Yaskawa INFORM job: A_ROOF_SIDE_0617_2_PAINT_42.JBI

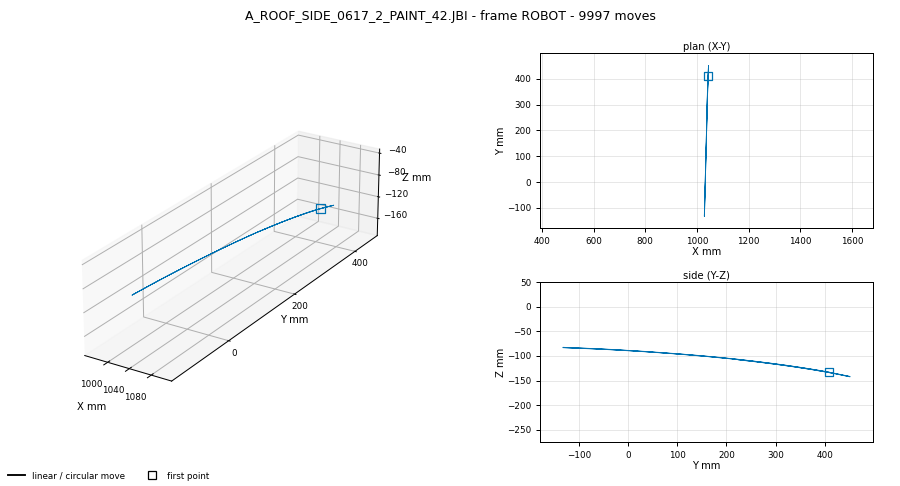
[picture p0: tool path of A_ROOF_SIDE_0617_2_PAINT_42.JBI in frame ROBOT, 9997 of 9997 moves have a stored position in this frame; points joined in program order, loops and branches not executed]
/JOB
//NAME A_ROOF_SIDE_0617_2_PAINT42
//POS
///NPOS 9997,0,0,0,0,0
///TOOL 1
///USER 0
///POSTYPE ROBOT
///RECTAN
///RCONF 1,0,0,0,0,0,0,0,0,0,0,0,0,0,0,0,0,0,0,0,0,0,0,0
C00000=1043.700,409.067,-132.998,174.418,43.875,158.706
C00001=1043.690,408.820,-132.952,174.408,43.868,158.704
C00002=1043.680,408.575,-132.906,174.398,43.862,158.701
C00003=1043.671,408.330,-132.861,174.389,43.855,158.699
C00004=1043.661,408.085,-132.816,174.379,43.848,158.696
C00005=1043.651,407.839,-132.770,174.370,43.842,158.694
C00006=1043.642,407.593,-132.725,174.361,43.835,158.691
C00007=1043.632,407.347,-132.680,174.352,43.829,158.689
C00008=1043.623,407.101,-132.635,174.342,43.822,158.686
C00009=1043.613,406.855,-132.589,174.333,43.816,158.684
C00010=1043.603,406.610,-132.544,174.325,43.809,158.681
C00011=1043.594,406.364,-132.499,174.315,43.802,158.679
C00012=1043.586,406.155,-132.460,174.308,43.797,158.677
C00013=1043.578,405.946,-132.422,174.300,43.791,158.674
C00014=1043.570,405.736,-132.384,174.292,43.786,158.672
C00015=1043.561,405.527,-132.345,174.284,43.780,158.670
C00016=1043.554,405.317,-132.307,174.277,43.775,158.668
C00017=1043.545,405.108,-132.268,174.269,43.770,158.666
C00018=1043.537,404.898,-132.230,174.261,43.764,158.664
C00019=1043.530,404.689,-132.192,174.254,43.759,158.662
C00020=1043.520,404.444,-132.147,174.244,43.753,158.660
C00021=1043.511,404.197,-132.102,174.235,43.746,158.657
C00022=1043.502,403.952,-132.058,174.226,43.740,158.655
C00023=1043.492,403.706,-132.013,174.218,43.733,158.652
C00024=1043.483,403.460,-131.968,174.209,43.727,158.650
C00025=1043.474,403.214,-131.923,174.200,43.721,158.648
C00026=1043.464,402.968,-131.879,174.191,43.715,158.645
C00027=1043.454,402.723,-131.834,174.183,43.708,158.643
C00028=1043.445,402.477,-131.790,174.174,43.702,158.640
C00029=1043.436,402.231,-131.745,174.164,43.696,158.638
C00030=1043.427,401.985,-131.701,174.156,43.690,158.636
C00031=1043.417,401.740,-131.656,174.147,43.684,158.634
C00032=1043.408,401.494,-131.612,174.138,43.678,158.631
C00033=1043.399,401.248,-131.568,174.130,43.671,158.629
C00034=1043.390,401.002,-131.524,174.121,43.666,158.627
C00035=1043.380,400.757,-131.479,174.112,43.660,158.624
C00036=1043.371,400.511,-131.435,174.104,43.653,158.622
C00037=1043.362,400.264,-131.391,174.096,43.648,158.620
C00038=1043.353,400.019,-131.347,174.086,43.641,158.617
C00039=1043.344,399.773,-131.303,174.079,43.635,158.615
C00040=1043.334,399.527,-131.259,174.070,43.630,158.613
C00041=1043.325,399.281,-131.215,174.062,43.623,158.611
C00042=1043.315,399.035,-131.171,174.053,43.618,158.609
C00043=1043.306,398.789,-131.127,174.045,43.612,158.606
C00044=1043.297,398.544,-131.083,174.036,43.606,158.604
C00045=1043.288,398.297,-131.040,174.028,43.600,158.602
C00046=1043.279,398.051,-130.996,174.019,43.594,158.600
C00047=1043.270,397.805,-130.952,174.012,43.588,158.598
C00048=1043.261,397.560,-130.908,174.003,43.583,158.595
C00049=1043.252,397.313,-130.865,173.995,43.577,158.593
C00050=1043.243,397.068,-130.821,173.986,43.571,158.591
C00051=1043.234,396.822,-130.777,173.978,43.565,158.589
C00052=1043.225,396.575,-130.734,173.970,43.559,158.587
C00053=1043.216,396.329,-130.690,173.962,43.554,158.584
C00054=1043.206,396.084,-130.647,173.953,43.548,158.582
C00055=1043.198,395.838,-130.604,173.945,43.542,158.580
C00056=1043.188,395.592,-130.560,173.937,43.536,158.578
C00057=1043.180,395.346,-130.517,173.929,43.531,158.576
C00058=1043.171,395.100,-130.474,173.921,43.525,158.574
C00059=1043.162,394.854,-130.430,173.913,43.519,158.572
C00060=1043.153,394.608,-130.387,173.905,43.514,158.570
C00061=1043.144,394.362,-130.344,173.897,43.508,158.568
C00062=1043.135,394.116,-130.300,173.889,43.502,158.565
C00063=1043.126,393.870,-130.258,173.880,43.497,158.563
C00064=1043.117,393.624,-130.215,173.873,43.491,158.561
C00065=1043.109,393.378,-130.172,173.865,43.486,158.559
C00066=1043.100,393.131,-130.128,173.856,43.480,158.557
C00067=1043.090,392.886,-130.086,173.849,43.475,158.555
C00068=1043.082,392.639,-130.043,173.841,43.469,158.553
C00069=1043.073,392.393,-130.000,173.833,43.464,158.551
C00070=1043.064,392.148,-129.957,173.825,43.458,158.549
C00071=1043.056,391.902,-129.914,173.817,43.453,158.547
C00072=1043.041,391.502,-129.844,173.805,43.444,158.544
C00073=1043.027,391.102,-129.775,173.792,43.435,158.540
C00074=1043.012,390.702,-129.706,173.780,43.426,158.537
C00075=1042.998,390.303,-129.637,173.767,43.418,158.534
C00076=1042.989,390.057,-129.594,173.759,43.413,158.532
C00077=1042.981,389.811,-129.551,173.752,43.407,158.530
C00078=1042.972,389.565,-129.509,173.744,43.402,158.528
C00079=1042.963,389.319,-129.466,173.737,43.397,158.526
C00080=1042.954,389.073,-129.424,173.729,43.391,158.524
C00081=1042.946,388.826,-129.381,173.722,43.386,158.522
C00082=1042.937,388.580,-129.339,173.713,43.381,158.520
C00083=1042.929,388.334,-129.297,173.706,43.376,158.519
C00084=1042.919,388.088,-129.254,173.698,43.371,158.517
C00085=1042.910,387.842,-129.213,173.691,43.365,158.515
C00086=1042.902,387.595,-129.170,173.683,43.360,158.513
C00087=1042.893,387.349,-129.128,173.676,43.355,158.511
C00088=1042.884,387.103,-129.086,173.669,43.350,158.509
C00089=1042.876,386.856,-129.044,173.661,43.345,158.507
C00090=1042.867,386.610,-129.002,173.654,43.340,158.505
C00091=1042.859,386.364,-128.961,173.646,43.334,158.503
C00092=1042.849,386.118,-128.918,173.639,43.330,158.502
C00093=1042.841,385.872,-128.876,173.632,43.324,158.500
C00094=1042.832,385.625,-128.834,173.624,43.319,158.498
C00095=1042.823,385.379,-128.793,173.617,43.315,158.496
C00096=1042.815,385.133,-128.751,173.609,43.309,158.494
C00097=1042.807,384.887,-128.709,173.602,43.304,158.492
C00098=1042.798,384.640,-128.667,173.595,43.300,158.490
C00099=1042.789,384.394,-128.625,173.588,43.295,158.489
C00100=1042.781,384.148,-128.584,173.580,43.289,158.487
C00101=1042.772,383.902,-128.542,173.573,43.284,158.485
C00102=1042.763,383.655,-128.500,173.566,43.280,158.483
C00103=1042.755,383.409,-128.459,173.558,43.275,158.481
C00104=1042.746,383.163,-128.418,173.551,43.270,158.480
C00105=1042.738,382.916,-128.375,173.545,43.265,158.478
C00106=1042.730,382.670,-128.334,173.538,43.260,158.476
C00107=1042.721,382.423,-128.293,173.530,43.255,158.474
C00108=1042.712,382.177,-128.251,173.523,43.250,158.472
C00109=1042.705,381.931,-128.209,173.516,43.245,158.471
C00110=1042.696,381.684,-128.168,173.508,43.241,158.469
C00111=1042.688,381.438,-128.127,173.501,43.236,158.467
C00112=1042.679,381.192,-128.085,173.495,43.231,158.465
C00113=1042.672,380.945,-128.044,173.488,43.226,158.464
C00114=1042.663,380.699,-128.002,173.480,43.221,158.462
C00115=1042.655,380.453,-127.962,173.473,43.217,158.460
C00116=1042.646,380.206,-127.920,173.466,43.212,158.458
C00117=1042.638,379.960,-127.879,173.460,43.207,158.457
C00118=1042.629,379.713,-127.837,173.453,43.202,158.455
C00119=1042.621,379.467,-127.797,173.446,43.198,158.453
C00120=1042.613,379.221,-127.756,173.438,43.193,158.451
C00121=1042.604,378.974,-127.714,173.432,43.188,158.450
C00122=1042.596,378.728,-127.674,173.425,43.183,158.448
C00123=1042.588,378.481,-127.633,173.418,43.178,158.446
C00124=1042.580,378.235,-127.592,173.411,43.174,158.445
C00125=1042.571,377.988,-127.551,173.405,43.170,158.443
C00126=1042.563,377.742,-127.510,173.398,43.165,158.441
C00127=1042.555,377.495,-127.470,173.391,43.160,158.440
C00128=1042.542,377.130,-127.409,173.380,43.154,158.437
C00129=1042.530,376.764,-127.349,173.370,43.147,158.435
C00130=1042.518,376.398,-127.288,173.360,43.140,158.432
C00131=1042.505,376.032,-127.228,173.351,43.133,158.430
C00132=1042.497,375.786,-127.187,173.344,43.128,158.428
C00133=1042.489,375.539,-127.146,173.337,43.124,158.427
C00134=1042.481,375.292,-127.106,173.331,43.120,158.425
C00135=1042.472,375.046,-127.066,173.324,43.115,158.423
C00136=1042.464,374.799,-127.026,173.317,43.111,158.422
C00137=1042.456,374.552,-126.985,173.311,43.106,158.420
C00138=1042.448,374.306,-126.944,173.304,43.102,158.419
C00139=1042.440,374.059,-126.904,173.298,43.098,158.417
C00140=1042.432,373.813,-126.863,173.291,43.093,158.416
C00141=1042.424,373.567,-126.823,173.284,43.089,158.414
C00142=1042.415,373.319,-126.783,173.278,43.084,158.412
C00143=1042.407,373.073,-126.743,173.271,43.080,158.411
C00144=1042.399,372.827,-126.702,173.265,43.076,158.409
C00145=1042.391,372.580,-126.662,173.258,43.071,158.408
C00146=1042.383,372.334,-126.621,173.252,43.067,158.406
C00147=1042.375,372.087,-126.581,173.245,43.062,158.404
C00148=1042.367,371.840,-126.541,173.239,43.058,158.403
C00149=1042.359,371.594,-126.501,173.232,43.054,158.401
C00150=1042.351,371.348,-126.461,173.226,43.050,158.400
C00151=1042.343,371.101,-126.421,173.219,43.045,158.398
C00152=1042.335,370.854,-126.381,173.213,43.041,158.397
C00153=1042.327,370.608,-126.340,173.206,43.037,158.395
C00154=1042.319,370.361,-126.301,173.200,43.032,158.394
C00155=1042.311,370.114,-126.261,173.193,43.028,158.392
C00156=1042.303,369.867,-126.222,173.188,43.024,158.391
C00157=1042.295,369.621,-126.182,173.181,43.020,158.389
C00158=1042.286,369.375,-126.142,173.175,43.016,158.388
C00159=1042.278,369.128,-126.102,173.169,43.011,158.386
C00160=1042.270,368.881,-126.063,173.162,43.007,158.385
C00161=1042.262,368.634,-126.023,173.156,43.003,158.383
C00162=1042.254,368.388,-125.983,173.149,42.999,158.382
C00163=1042.246,368.141,-125.943,173.144,42.995,158.380
C00164=1042.238,367.894,-125.904,173.137,42.991,158.379
C00165=1042.230,367.647,-125.864,173.131,42.987,158.377
C00166=1042.221,367.401,-125.825,173.125,42.983,158.376
C00167=1042.214,367.154,-125.785,173.118,42.978,158.374
C00168=1042.206,366.907,-125.747,173.112,42.974,158.373
C00169=1042.198,366.660,-125.707,173.107,42.970,158.371
C00170=1042.190,366.414,-125.667,173.100,42.966,158.370
C00171=1042.182,366.167,-125.628,173.094,42.962,158.368
C00172=1042.174,365.920,-125.588,173.088,42.958,158.367
C00173=1042.166,365.673,-125.548,173.081,42.954,158.366
C00174=1042.158,365.427,-125.510,173.076,42.950,158.364
C00175=1042.151,365.180,-125.470,173.070,42.946,158.363
C00176=1042.142,364.933,-125.431,173.063,42.942,158.361
C00177=1042.135,364.686,-125.392,173.057,42.938,158.360
C00178=1042.127,364.440,-125.353,173.051,42.934,158.358
C00179=1042.119,364.193,-125.313,173.045,42.930,158.357
C00180=1042.111,363.946,-125.274,173.039,42.926,158.356
C00181=1042.104,363.699,-125.235,173.033,42.922,158.354
C00182=1042.096,363.452,-125.196,173.027,42.918,158.353
C00183=1042.088,363.205,-125.156,173.021,42.914,158.351
C00184=1042.077,362.859,-125.102,173.012,42.909,158.349
C00185=1042.066,362.513,-125.047,173.004,42.904,158.348
C00186=1042.056,362.168,-124.992,172.997,42.898,158.346
C00187=1042.045,361.821,-124.938,172.988,42.893,158.344
C00188=1042.037,361.574,-124.899,172.981,42.889,158.342
C00189=1042.028,361.327,-124.860,172.976,42.885,158.341
C00190=1042.021,361.081,-124.822,172.970,42.881,158.340
C00191=1042.013,360.833,-124.782,172.964,42.877,158.338
C00192=1042.006,360.587,-124.744,172.959,42.873,158.337
C00193=1041.997,360.340,-124.705,172.952,42.870,158.335
C00194=1041.989,360.093,-124.666,172.946,42.866,158.334
C00195=1041.982,359.847,-124.628,172.941,42.862,158.333
C00196=1041.974,359.599,-124.589,172.935,42.859,158.332
C00197=1041.967,359.353,-124.550,172.929,42.855,158.330
C00198=1041.959,359.105,-124.512,172.923,42.851,158.329
C00199=1041.951,358.859,-124.474,172.917,42.847,158.328
C00200=1041.943,358.612,-124.435,172.911,42.843,158.326
C00201=1041.935,358.365,-124.397,172.906,42.840,158.325
C00202=1041.927,358.118,-124.358,172.900,42.836,158.324
C00203=1041.920,357.871,-124.320,172.895,42.833,158.322
C00204=1041.912,357.624,-124.281,172.889,42.829,158.321
C00205=1041.905,357.377,-124.242,172.883,42.825,158.320
C00206=1041.897,357.131,-124.204,172.877,42.822,158.318
C00207=1041.889,356.884,-124.166,172.871,42.818,158.317
C00208=1041.882,356.636,-124.128,172.866,42.814,158.316
C00209=1041.874,356.389,-124.089,172.860,42.810,158.314
C00210=1041.866,356.143,-124.051,172.854,42.807,158.313
C00211=1041.859,355.896,-124.013,172.849,42.803,158.312
C00212=1041.851,355.648,-123.975,172.843,42.800,158.311
C00213=1041.843,355.402,-123.937,172.838,42.796,158.309
C00214=1041.835,355.155,-123.898,172.832,42.793,158.308
C00215=1041.828,354.908,-123.861,172.827,42.789,158.307
C00216=1041.820,354.661,-123.822,172.821,42.786,158.306
C00217=1041.812,354.413,-123.785,172.816,42.782,158.305
C00218=1041.804,354.167,-123.747,172.810,42.779,158.303
C00219=1041.797,353.920,-123.709,172.804,42.775,158.302
C00220=1041.789,353.673,-123.671,172.799,42.771,158.301
C00221=1041.781,353.425,-123.633,172.792,42.768,158.299
C00222=1041.774,353.179,-123.595,172.787,42.765,158.298
C00223=1041.767,352.932,-123.557,172.781,42.761,158.297
C00224=1041.759,352.685,-123.519,172.776,42.758,158.296
C00225=1041.751,352.437,-123.481,172.771,42.754,158.295
C00226=1041.744,352.191,-123.443,172.766,42.751,158.293
C00227=1041.736,351.944,-123.406,172.760,42.747,158.292
C00228=1041.729,351.697,-123.368,172.755,42.744,158.291
C00229=1041.722,351.450,-123.330,172.749,42.740,158.290
C00230=1041.713,351.203,-123.293,172.744,42.737,158.288
C00231=1041.706,350.955,-123.255,172.738,42.733,158.287
C00232=1041.699,350.708,-123.217,172.733,42.730,158.286
C00233=1041.691,350.462,-123.179,172.727,42.726,158.285
C00234=1041.684,350.215,-123.142,172.722,42.723,158.284
C00235=1041.677,349.968,-123.104,172.717,42.720,158.283
C00236=1041.669,349.720,-123.067,172.711,42.717,158.281
C00237=1041.661,349.473,-123.029,172.706,42.713,158.280
C00238=1041.653,349.226,-122.992,172.700,42.710,158.279
C00239=1041.646,348.979,-122.954,172.695,42.706,158.278
C00240=1041.636,348.639,-122.903,172.688,42.702,158.276
C00241=1041.625,348.299,-122.852,172.681,42.697,158.275
C00242=1041.615,347.958,-122.800,172.673,42.693,158.273
C00243=1041.604,347.618,-122.749,172.666,42.688,158.271
C00244=1041.596,347.371,-122.712,172.660,42.685,158.270
C00245=1041.589,347.124,-122.674,172.655,42.682,158.269
C00246=1041.582,346.877,-122.637,172.650,42.679,158.268
C00247=1041.574,346.630,-122.600,172.644,42.675,158.267
C00248=1041.567,346.383,-122.562,172.640,42.672,158.266
C00249=1041.560,346.135,-122.526,172.634,42.669,158.264
C00250=1041.552,345.888,-122.489,172.629,42.666,158.263
C00251=1041.545,345.641,-122.451,172.624,42.662,158.262
C00252=1041.537,345.394,-122.414,172.618,42.659,158.261
C00253=1041.530,345.146,-122.377,172.613,42.656,158.260
C00254=1041.522,344.899,-122.340,172.609,42.653,158.259
C00255=1041.515,344.653,-122.303,172.603,42.649,158.258
C00256=1041.508,344.405,-122.266,172.598,42.646,158.257
C00257=1041.500,344.159,-122.229,172.592,42.643,158.255
C00258=1041.493,343.911,-122.192,172.587,42.640,158.254
C00259=1041.485,343.664,-122.156,172.583,42.637,158.253
C00260=1041.478,343.417,-122.118,172.577,42.634,158.252
C00261=1041.471,343.169,-122.081,172.572,42.631,158.251
C00262=1041.463,342.922,-122.044,172.567,42.628,158.250
C00263=1041.457,342.675,-122.008,172.562,42.624,158.249
C00264=1041.449,342.428,-121.971,172.557,42.621,158.248
C00265=1041.442,342.181,-121.934,172.552,42.618,158.247
C00266=1041.434,341.934,-121.897,172.546,42.615,158.245
C00267=1041.427,341.686,-121.861,172.542,42.612,158.244
C00268=1041.419,341.439,-121.824,172.537,42.609,158.243
C00269=1041.412,341.193,-121.788,172.532,42.606,158.242
C00270=1041.404,340.945,-121.752,172.526,42.603,158.241
C00271=1041.397,340.697,-121.715,172.522,42.599,158.240
C00272=1041.389,340.450,-121.678,172.517,42.596,158.239
C00273=1041.381,340.203,-121.642,172.511,42.594,158.238
C00274=1041.375,339.956,-121.605,172.506,42.591,158.237
C00275=1041.367,339.709,-121.569,172.502,42.588,158.236
C00276=1041.360,339.461,-121.533,172.496,42.585,158.235
C00277=1041.352,339.214,-121.496,172.491,42.582,158.234
C00278=1041.345,338.967,-121.459,172.487,42.579,158.233
C00279=1041.338,338.720,-121.423,172.482,42.576,158.232
C00280=1041.330,338.472,-121.387,172.476,42.573,158.231
C00281=1041.324,338.225,-121.350,172.472,42.570,158.230
C00282=1041.316,337.978,-121.314,172.467,42.567,158.229
C00283=1041.308,337.730,-121.278,172.462,42.564,158.228
C00284=1041.301,337.484,-121.242,172.457,42.561,158.227
C00285=1041.294,337.236,-121.205,172.452,42.558,158.225
C00286=1041.287,336.988,-121.169,172.447,42.555,158.224
C00287=1041.280,336.742,-121.133,172.443,42.552,158.223
C00288=1041.272,336.494,-121.097,172.437,42.549,158.222
C00289=1041.266,336.247,-121.061,172.432,42.546,158.221
C00290=1041.258,336.000,-121.024,172.428,42.543,158.220
C00291=1041.250,335.752,-120.988,172.423,42.540,158.219
C00292=1041.243,335.506,-120.952,172.419,42.538,158.218
C00293=1041.237,335.257,-120.916,172.413,42.535,158.217
C00294=1041.230,335.010,-120.880,172.408,42.532,158.216
C00295=1041.222,334.763,-120.844,172.404,42.529,158.215
C00296=1041.211,334.419,-120.795,172.397,42.525,158.214
C00297=1041.201,334.076,-120.745,172.390,42.521,158.212
C00298=1041.191,333.732,-120.695,172.384,42.517,158.211
C00299=1041.182,333.388,-120.645,172.377,42.514,158.210
C00300=1041.174,333.140,-120.609,172.372,42.511,158.209
C00301=1041.167,332.893,-120.574,172.368,42.507,158.208
C00302=1041.159,332.646,-120.537,172.363,42.505,158.207
C00303=1041.153,332.398,-120.502,172.357,42.502,158.206
C00304=1041.145,332.151,-120.466,172.353,42.499,158.205
C00305=1041.138,331.903,-120.431,172.348,42.497,158.204
C00306=1041.131,331.656,-120.395,172.344,42.494,158.203
C00307=1041.124,331.409,-120.359,172.339,42.491,158.202
C00308=1041.116,331.161,-120.323,172.335,42.488,158.201
C00309=1041.109,330.914,-120.288,172.329,42.485,158.200
C00310=1041.102,330.667,-120.252,172.325,42.483,158.199
C00311=1041.095,330.419,-120.217,172.320,42.480,158.198
C00312=1041.088,330.172,-120.181,172.316,42.477,158.197
C00313=1041.080,329.924,-120.145,172.311,42.474,158.196
C00314=1041.073,329.677,-120.110,172.307,42.472,158.195
C00315=1041.067,329.430,-120.074,172.302,42.469,158.194
C00316=1041.059,329.182,-120.040,172.297,42.467,158.193
C00317=1041.051,328.936,-120.004,172.292,42.464,158.192
C00318=1041.045,328.688,-119.969,172.288,42.461,158.192
C00319=1041.037,328.440,-119.933,172.283,42.459,158.191
C00320=1041.030,328.193,-119.899,172.279,42.456,158.190
C00321=1041.022,327.945,-119.863,172.274,42.453,158.189
C00322=1041.015,327.698,-119.828,172.270,42.451,158.188
C00323=1041.008,327.451,-119.793,172.265,42.448,158.187
C00324=1041.000,327.203,-119.757,172.261,42.445,158.186
C00325=1040.993,326.956,-119.723,172.256,42.443,158.185
C00326=1040.986,326.709,-119.687,172.251,42.440,158.184
C00327=1040.978,326.461,-119.653,172.246,42.438,158.183
C00328=1040.971,326.214,-119.617,172.242,42.435,158.182
C00329=1040.964,325.967,-119.583,172.237,42.433,158.181
C00330=1040.956,325.718,-119.547,172.233,42.430,158.181
C00331=1040.950,325.471,-119.512,172.228,42.428,158.180
C00332=1040.942,325.224,-119.478,172.224,42.425,158.179
C00333=1040.935,324.977,-119.443,172.219,42.423,158.178
C00334=1040.928,324.728,-119.408,172.215,42.420,158.177
C00335=1040.921,324.481,-119.373,172.211,42.417,158.176
C00336=1040.913,324.234,-119.339,172.206,42.415,158.175
C00337=1040.907,323.987,-119.304,172.202,42.412,158.174
C00338=1040.898,323.739,-119.269,172.197,42.410,158.173
C00339=1040.892,323.491,-119.234,172.193,42.408,158.173
C00340=1040.885,323.244,-119.198,172.188,42.405,158.172
C00341=1040.878,322.996,-119.165,172.184,42.403,158.171
C00342=1040.871,322.749,-119.129,172.180,42.400,158.170
C00343=1040.863,322.502,-119.095,172.174,42.398,158.169
C00344=1040.856,322.254,-119.059,172.170,42.395,158.168
C00345=1040.849,322.006,-119.026,172.166,42.392,158.167
C00346=1040.842,321.759,-118.990,172.161,42.390,158.166
C00347=1040.835,321.512,-118.956,172.157,42.387,158.166
C00348=1040.828,321.264,-118.921,172.152,42.385,158.165
C00349=1040.821,321.017,-118.887,172.148,42.382,158.164
C00350=1040.814,320.769,-118.852,172.144,42.380,158.163
C00351=1040.807,320.522,-118.818,172.139,42.377,158.162
C00352=1040.797,320.173,-118.768,172.134,42.374,158.161
C00353=1040.787,319.825,-118.720,172.127,42.370,158.160
C00354=1040.777,319.476,-118.671,172.121,42.367,158.158
C00355=1040.767,319.127,-118.623,172.115,42.363,158.157
C00356=1040.760,318.879,-118.588,172.110,42.362,158.156
C00357=1040.753,318.632,-118.554,172.106,42.359,158.156
C00358=1040.746,318.384,-118.519,172.102,42.357,158.155
C00359=1040.739,318.137,-118.485,172.097,42.354,158.154
C00360=1040.732,317.889,-118.450,172.093,42.352,158.153
C00361=1040.725,317.642,-118.416,172.089,42.349,158.152
C00362=1040.718,317.394,-118.381,172.085,42.347,158.151
C00363=1040.711,317.147,-118.347,172.080,42.344,158.150
C00364=1040.704,316.899,-118.312,172.076,42.342,158.150
C00365=1040.697,316.651,-118.279,172.072,42.340,158.149
C00366=1040.691,316.405,-118.244,172.068,42.337,158.148
C00367=1040.684,316.157,-118.210,172.063,42.335,158.147
C00368=1040.677,315.909,-118.176,172.059,42.332,158.146
C00369=1040.670,315.662,-118.141,172.055,42.330,158.145
C00370=1040.663,315.414,-118.107,172.052,42.328,158.145
C00371=1040.656,315.166,-118.073,172.046,42.326,158.144
C00372=1040.649,314.919,-118.038,172.042,42.323,158.143
C00373=1040.643,314.672,-118.004,172.038,42.320,158.142
C00374=1040.636,314.424,-117.970,172.034,42.318,158.141
C00375=1040.629,314.176,-117.936,172.030,42.316,158.141
C00376=1040.622,313.929,-117.901,172.026,42.314,158.140
C00377=1040.615,313.681,-117.867,172.022,42.311,158.139
C00378=1040.609,313.434,-117.833,172.018,42.309,158.138
C00379=1040.601,313.187,-117.800,172.014,42.307,158.137
C00380=1040.595,312.939,-117.765,172.010,42.304,158.137
C00381=1040.588,312.691,-117.731,172.005,42.302,158.136
C00382=1040.582,312.444,-117.697,172.001,42.300,158.135
C00383=1040.574,312.197,-117.663,171.997,42.297,158.134
C00384=1040.567,311.949,-117.629,171.993,42.295,158.133
C00385=1040.560,311.701,-117.596,171.989,42.293,158.133
C00386=1040.553,311.453,-117.562,171.984,42.290,158.132
C00387=1040.547,311.206,-117.529,171.980,42.288,158.131
C00388=1040.539,310.958,-117.495,171.976,42.286,158.130
C00389=1040.532,310.711,-117.461,171.972,42.284,158.129
C00390=1040.524,310.463,-117.428,171.968,42.282,158.129
C00391=1040.517,310.216,-117.394,171.963,42.280,158.128
C00392=1040.511,309.968,-117.361,171.960,42.278,158.127
C00393=1040.504,309.720,-117.327,171.956,42.276,158.126
C00394=1040.496,309.473,-117.294,171.952,42.273,158.126
C00395=1040.489,309.225,-117.260,171.947,42.271,158.125
C00396=1040.483,308.978,-117.227,171.943,42.269,158.124
C00397=1040.476,308.730,-117.193,171.939,42.267,158.123
C00398=1040.468,308.482,-117.160,171.935,42.265,158.123
C00399=1040.460,308.235,-117.126,171.931,42.262,158.122
C00400=1040.454,307.987,-117.093,171.928,42.260,158.121
C00401=1040.447,307.740,-117.060,171.923,42.259,158.120
C00402=1040.440,307.491,-117.026,171.919,42.256,158.120
C00403=1040.433,307.244,-116.993,171.915,42.254,158.119
C00404=1040.426,306.997,-116.960,171.911,42.252,158.118
C00405=1040.419,306.749,-116.927,171.907,42.250,158.117
C00406=1040.412,306.502,-116.893,171.903,42.248,158.117
C00407=1040.405,306.253,-116.860,171.899,42.246,158.116
C00408=1040.396,305.910,-116.813,171.893,42.243,158.115
C00409=1040.386,305.566,-116.767,171.888,42.240,158.114
C00410=1040.377,305.222,-116.721,171.883,42.237,158.113
C00411=1040.367,304.878,-116.675,171.877,42.234,158.112
C00412=1040.359,304.631,-116.642,171.873,42.232,158.111
C00413=1040.352,304.383,-116.609,171.869,42.230,158.110
C00414=1040.346,304.136,-116.576,171.865,42.227,158.110
C00415=1040.339,303.887,-116.542,171.861,42.225,158.109
C00416=1040.332,303.639,-116.509,171.857,42.223,158.108
C00417=1040.326,303.392,-116.476,171.854,42.222,158.107
C00418=1040.318,303.144,-116.443,171.850,42.219,158.107
C00419=1040.311,302.897,-116.410,171.846,42.217,158.106
C00420=1040.304,302.649,-116.377,171.842,42.215,158.105
C00421=1040.298,302.401,-116.344,171.838,42.213,158.105
C00422=1040.291,302.154,-116.310,171.834,42.211,158.104
C00423=1040.284,301.906,-116.278,171.830,42.209,158.103
C00424=1040.277,301.658,-116.245,171.826,42.207,158.102
C00425=1040.271,301.411,-116.212,171.823,42.205,158.102
C00426=1040.264,301.164,-116.179,171.819,42.203,158.101
C00427=1040.257,300.915,-116.146,171.815,42.201,158.100
C00428=1040.250,300.668,-116.114,171.810,42.199,158.100
C00429=1040.243,300.420,-116.080,171.806,42.196,158.099
C00430=1040.237,300.173,-116.047,171.802,42.194,158.098
C00431=1040.230,299.924,-116.014,171.799,42.192,158.097
C00432=1040.223,299.677,-115.982,171.795,42.190,158.097
C00433=1040.216,299.430,-115.949,171.791,42.188,158.096
C00434=1040.210,299.181,-115.916,171.788,42.186,158.095
C00435=1040.203,298.934,-115.883,171.784,42.184,158.095
C00436=1040.197,298.686,-115.850,171.781,42.182,158.094
C00437=1040.189,298.439,-115.817,171.777,42.180,158.093
C00438=1040.183,298.191,-115.784,171.773,42.178,158.092
C00439=1040.176,297.944,-115.752,171.769,42.176,158.092
C00440=1040.170,297.695,-115.719,171.765,42.174,158.091
C00441=1040.163,297.448,-115.686,171.761,42.172,158.090
C00442=1040.156,297.200,-115.654,171.758,42.170,158.090
C00443=1040.149,296.952,-115.621,171.754,42.168,158.089
C00444=1040.143,296.704,-115.588,171.750,42.166,158.088
C00445=1040.136,296.457,-115.556,171.746,42.164,158.088
C00446=1040.129,296.209,-115.523,171.742,42.162,158.087
C00447=1040.123,295.961,-115.490,171.739,42.160,158.086
C00448=1040.117,295.714,-115.457,171.735,42.158,158.085
C00449=1040.109,295.466,-115.425,171.731,42.156,158.085
C00450=1040.103,295.218,-115.393,171.727,42.154,158.084
C00451=1040.096,294.970,-115.360,171.723,42.152,158.083
C00452=1040.090,294.723,-115.328,171.721,42.150,158.083
C00453=1040.082,294.475,-115.295,171.717,42.148,158.082
C00454=1040.076,294.227,-115.262,171.713,42.146,158.081
C00455=1040.069,293.979,-115.231,171.709,42.144,158.081
C00456=1040.063,293.732,-115.198,171.705,42.143,158.080
C00457=1040.055,293.484,-115.166,171.702,42.141,158.079
C00458=1040.049,293.236,-115.133,171.698,42.139,158.079
C00459=1040.042,292.988,-115.102,171.694,42.137,158.078
C00460=1040.034,292.740,-115.069,171.690,42.135,158.077
C00461=1040.028,292.492,-115.037,171.687,42.134,158.077
C00462=1040.021,292.245,-115.005,171.683,42.132,158.076
C00463=1040.014,291.997,-114.973,171.679,42.130,158.075
C00464=1040.006,291.669,-114.931,171.675,42.127,158.075
C00465=1039.996,291.342,-114.888,171.670,42.125,158.074
C00466=1039.987,291.015,-114.845,171.665,42.122,158.073
C00467=1039.979,290.687,-114.803,171.660,42.120,158.072
C00468=1039.972,290.440,-114.771,171.656,42.118,158.071
C00469=1039.966,290.192,-114.739,171.653,42.116,158.071
C00470=1039.959,289.944,-114.707,171.650,42.114,158.070
C00471=1039.951,289.696,-114.675,171.646,42.112,158.069
C00472=1039.944,289.448,-114.643,171.642,42.110,158.069
C00473=1039.938,289.200,-114.611,171.639,42.109,158.068
C00474=1039.931,288.953,-114.579,171.635,42.107,158.068
C00475=1039.924,288.705,-114.547,171.631,42.105,158.067
C00476=1039.918,288.457,-114.516,171.627,42.104,158.066
C00477=1039.911,288.209,-114.483,171.625,42.101,158.066
C00478=1039.904,287.961,-114.451,171.621,42.099,158.065
C00479=1039.897,287.714,-114.419,171.617,42.098,158.064
C00480=1039.890,287.466,-114.388,171.613,42.096,158.064
C00481=1039.884,287.218,-114.356,171.610,42.094,158.063
C00482=1039.878,286.970,-114.324,171.606,42.093,158.062
C00483=1039.871,286.722,-114.292,171.603,42.091,158.062
C00484=1039.864,286.475,-114.261,171.599,42.089,158.061
C00485=1039.857,286.226,-114.229,171.596,42.087,158.061
C00486=1039.850,285.978,-114.198,171.592,42.085,158.060
C00487=1039.843,285.731,-114.165,171.588,42.084,158.059
C00488=1039.836,285.483,-114.134,171.585,42.082,158.059
C00489=1039.829,285.235,-114.103,171.582,42.080,158.058
C00490=1039.823,284.987,-114.071,171.578,42.078,158.058
C00491=1039.816,284.739,-114.040,171.575,42.077,158.057
C00492=1039.809,284.491,-114.008,171.571,42.075,158.056
C00493=1039.802,284.243,-113.977,171.567,42.074,158.056
C00494=1039.796,283.995,-113.945,171.564,42.071,158.055
C00495=1039.789,283.747,-113.914,171.561,42.070,158.055
C00496=1039.782,283.500,-113.883,171.557,42.068,158.054
C00497=1039.775,283.252,-113.850,171.553,42.066,158.053
C00498=1039.768,283.004,-113.819,171.551,42.065,158.053
C00499=1039.761,282.756,-113.787,171.547,42.063,158.052
C00500=1039.754,282.508,-113.756,171.543,42.061,158.051
C00501=1039.748,282.260,-113.724,171.540,42.059,158.051
C00502=1039.741,282.012,-113.693,171.537,42.058,158.050
C00503=1039.735,281.764,-113.662,171.533,42.056,158.050
C00504=1039.728,281.516,-113.631,171.530,42.054,158.049
C00505=1039.722,281.268,-113.600,171.526,42.053,158.049
C00506=1039.715,281.021,-113.568,171.523,42.051,158.048
C00507=1039.708,280.773,-113.537,171.520,42.049,158.047
C00508=1039.702,280.525,-113.505,171.516,42.047,158.047
C00509=1039.695,280.277,-113.474,171.512,42.046,158.046
C00510=1039.688,280.029,-113.443,171.509,42.044,158.045
C00511=1039.681,279.781,-113.411,171.506,42.042,158.045
C00512=1039.675,279.533,-113.380,171.502,42.040,158.044
C00513=1039.668,279.285,-113.349,171.499,42.039,158.044
C00514=1039.662,279.037,-113.318,171.496,42.037,158.043
C00515=1039.655,278.789,-113.286,171.492,42.036,158.043
C00516=1039.647,278.541,-113.255,171.488,42.034,158.042
C00517=1039.641,278.293,-113.225,171.486,42.032,158.041
C00518=1039.634,278.045,-113.193,171.482,42.031,158.041
C00519=1039.628,277.798,-113.162,171.478,42.029,158.040
C00520=1039.618,277.482,-113.123,171.474,42.027,158.039
C00521=1039.610,277.166,-113.083,171.470,42.025,158.039
C00522=1039.602,276.851,-113.043,171.466,42.023,158.038
C00523=1039.594,276.535,-113.005,171.462,42.020,158.037
C00524=1039.586,276.287,-112.974,171.458,42.019,158.037
C00525=1039.580,276.040,-112.942,171.455,42.017,158.036
C00526=1039.573,275.791,-112.912,171.451,42.016,158.036
C00527=1039.566,275.544,-112.881,171.448,42.014,158.035
C00528=1039.560,275.296,-112.850,171.445,42.012,158.034
C00529=1039.553,275.048,-112.819,171.441,42.011,158.034
C00530=1039.547,274.799,-112.788,171.438,42.009,158.033
C00531=1039.539,274.552,-112.757,171.435,42.007,158.033
C00532=1039.533,274.303,-112.727,171.432,42.006,158.032
C00533=1039.527,274.056,-112.696,171.428,42.004,158.032
C00534=1039.520,273.808,-112.665,171.425,42.003,158.031
C00535=1039.513,273.560,-112.634,171.422,42.001,158.030
C00536=1039.506,273.311,-112.603,171.419,42.000,158.030
C00537=1039.499,273.064,-112.572,171.415,41.998,158.029
C00538=1039.493,272.815,-112.542,171.412,41.996,158.029
C00539=1039.486,272.568,-112.511,171.409,41.995,158.028
C00540=1039.479,272.320,-112.481,171.405,41.993,158.028
C00541=1039.473,272.071,-112.450,171.402,41.991,158.027
C00542=1039.465,271.824,-112.419,171.399,41.990,158.027
C00543=1039.460,271.576,-112.389,171.396,41.988,158.026
C00544=1039.453,271.327,-112.358,171.392,41.987,158.025
C00545=1039.446,271.080,-112.327,171.389,41.985,158.025
C00546=1039.439,270.831,-112.296,171.386,41.983,158.024
C00547=1039.433,270.584,-112.267,171.382,41.982,158.024
C00548=1039.426,270.335,-112.236,171.379,41.980,158.023
C00549=1039.419,270.087,-112.205,171.376,41.979,158.023
C00550=1039.412,269.839,-112.174,171.373,41.977,158.022
C00551=1039.406,269.591,-112.145,171.370,41.976,158.022
C00552=1039.399,269.343,-112.114,171.366,41.974,158.021
C00553=1039.392,269.095,-112.084,171.363,41.973,158.020
C00554=1039.386,268.847,-112.052,171.360,41.971,158.020
C00555=1039.379,268.599,-112.023,171.356,41.970,158.019
C00556=1039.373,268.351,-111.992,171.354,41.968,158.019
C00557=1039.365,268.103,-111.962,171.350,41.967,158.018
C00558=1039.359,267.855,-111.932,171.348,41.965,158.018
C00559=1039.352,267.606,-111.901,171.344,41.964,158.017
C00560=1039.345,267.358,-111.871,171.340,41.962,158.017
C00561=1039.339,267.110,-111.841,171.338,41.960,158.016
C00562=1039.332,266.862,-111.811,171.334,41.959,158.016
C00563=1039.325,266.614,-111.781,171.332,41.957,158.015
C00564=1039.319,266.366,-111.750,171.328,41.956,158.015
C00565=1039.312,266.118,-111.720,171.325,41.954,158.014
C00566=1039.305,265.870,-111.690,171.322,41.953,158.014
C00567=1039.299,265.622,-111.660,171.319,41.951,158.013
C00568=1039.292,265.374,-111.629,171.316,41.950,158.013
C00569=1039.285,265.126,-111.599,171.312,41.948,158.012
C00570=1039.279,264.878,-111.569,171.309,41.947,158.012
C00571=1039.272,264.630,-111.539,171.306,41.945,158.011
C00572=1039.265,264.382,-111.509,171.303,41.944,158.011
C00573=1039.259,264.133,-111.478,171.300,41.943,158.010
C00574=1039.252,263.885,-111.448,171.297,41.941,158.009
C00575=1039.245,263.638,-111.419,171.293,41.940,158.009
C00576=1039.238,263.326,-111.381,171.290,41.938,158.008
C00577=1039.229,263.016,-111.343,171.286,41.936,158.008
C00578=1039.220,262.704,-111.306,171.282,41.933,158.007
C00579=1039.212,262.393,-111.268,171.278,41.931,158.006
C00580=1039.205,262.146,-111.238,171.275,41.930,158.006
C00581=1039.198,261.897,-111.208,171.272,41.929,158.005
C00582=1039.192,261.650,-111.178,171.269,41.927,158.005
C00583=1039.185,261.401,-111.149,171.266,41.926,158.004
C00584=1039.178,261.153,-111.119,171.263,41.925,158.004
C00585=1039.171,260.905,-111.089,171.260,41.923,158.003
C00586=1039.164,260.657,-111.060,171.256,41.922,158.003
C00587=1039.158,260.409,-111.030,171.254,41.920,158.002
C00588=1039.151,260.160,-111.000,171.250,41.919,158.002
C00589=1039.144,259.912,-110.970,171.248,41.917,158.001
C00590=1039.137,259.664,-110.941,171.244,41.916,158.001
C00591=1039.130,259.416,-110.911,171.242,41.915,158.000
C00592=1039.124,259.168,-110.881,171.238,41.914,158.000
C00593=1039.116,258.920,-110.853,171.235,41.912,157.999
C00594=1039.110,258.672,-110.823,171.232,41.911,157.999
C00595=1039.103,258.423,-110.793,171.229,41.909,157.998
C00596=1039.096,258.176,-110.764,171.226,41.908,157.998
C00597=1039.089,257.927,-110.734,171.223,41.907,157.997
C00598=1039.083,257.679,-110.704,171.220,41.905,157.997
C00599=1039.076,257.431,-110.675,171.217,41.904,157.996
C00600=1039.069,257.183,-110.645,171.214,41.902,157.996
C00601=1039.063,256.934,-110.616,171.211,41.901,157.995
C00602=1039.056,256.687,-110.586,171.208,41.900,157.995
C00603=1039.049,256.438,-110.557,171.205,41.898,157.994
C00604=1039.042,256.191,-110.528,171.202,41.897,157.994
C00605=1039.035,255.942,-110.498,171.199,41.895,157.993
C00606=1039.029,255.694,-110.469,171.196,41.894,157.993
C00607=1039.022,255.445,-110.439,171.193,41.892,157.992
C00608=1039.015,255.197,-110.410,171.190,41.891,157.992
C00609=1039.008,254.949,-110.380,171.187,41.890,157.992
C00610=1039.002,254.701,-110.351,171.184,41.888,157.991
C00611=1038.995,254.452,-110.321,171.182,41.887,157.991
C00612=1038.989,254.205,-110.292,171.178,41.885,157.990
C00613=1038.982,253.957,-110.263,171.175,41.884,157.990
C00614=1038.975,253.708,-110.234,171.172,41.883,157.989
C00615=1038.968,253.460,-110.205,171.169,41.882,157.989
C00616=1038.961,253.212,-110.175,171.166,41.880,157.988
C00617=1038.955,252.964,-110.146,171.163,41.879,157.988
C00618=1038.949,252.715,-110.117,171.161,41.877,157.987
C00619=1038.942,252.467,-110.086,171.157,41.876,157.987
C00620=1038.935,252.219,-110.057,171.155,41.875,157.986
C00621=1038.929,251.970,-110.028,171.152,41.873,157.986
C00622=1038.922,251.722,-110.000,171.148,41.872,157.985
C00623=1038.915,251.474,-109.970,171.146,41.870,157.985
C00624=1038.908,251.226,-109.940,171.142,41.869,157.984
C00625=1038.902,250.978,-109.911,171.140,41.868,157.984
C00626=1038.896,250.730,-109.882,171.137,41.866,157.983
C00627=1038.889,250.481,-109.853,171.134,41.865,157.983
C00628=1038.883,250.233,-109.824,171.131,41.863,157.982
C00629=1038.875,249.986,-109.795,171.129,41.862,157.982
C00630=1038.868,249.737,-109.765,171.125,41.861,157.981
C00631=1038.862,249.489,-109.736,171.123,41.859,157.981
C00632=1038.854,249.176,-109.699,171.119,41.857,157.980
C00633=1038.846,248.864,-109.663,171.115,41.856,157.980
C00634=1038.838,248.551,-109.627,171.111,41.854,157.979
C00635=1038.829,248.239,-109.590,171.108,41.852,157.979
C00636=1038.823,247.991,-109.561,171.105,41.851,157.978
C00637=1038.816,247.743,-109.532,171.103,41.849,157.978
C00638=1038.810,247.495,-109.503,171.099,41.848,157.977
C00639=1038.803,247.246,-109.473,171.097,41.846,157.977
C00640=1038.797,246.998,-109.444,171.094,41.845,157.976
C00641=1038.791,246.750,-109.415,171.092,41.844,157.976
C00642=1038.784,246.502,-109.387,171.088,41.842,157.975
C00643=1038.777,246.254,-109.358,171.085,41.841,157.975
C00644=1038.771,246.005,-109.328,171.083,41.839,157.974
C00645=1038.764,245.757,-109.299,171.079,41.838,157.974
C00646=1038.758,245.509,-109.270,171.077,41.837,157.973
C00647=1038.752,245.261,-109.241,171.074,41.835,157.973
C00648=1038.745,245.013,-109.213,171.072,41.834,157.972
C00649=1038.738,244.764,-109.183,171.068,41.832,157.972
C00650=1038.732,244.516,-109.154,171.066,41.831,157.971
C00651=1038.725,244.267,-109.127,171.063,41.830,157.971
C00652=1038.719,244.019,-109.097,171.061,41.828,157.970
C00653=1038.711,243.771,-109.069,171.057,41.827,157.970
C00654=1038.705,243.523,-109.040,171.055,41.826,157.970
C00655=1038.698,243.275,-109.011,171.052,41.824,157.969
C00656=1038.692,243.026,-108.983,171.049,41.823,157.969
C00657=1038.686,242.778,-108.954,171.046,41.822,157.968
C00658=1038.678,242.529,-108.925,171.044,41.820,157.968
C00659=1038.672,242.281,-108.896,171.041,41.819,157.967
C00660=1038.665,242.033,-108.868,171.038,41.818,157.967
C00661=1038.659,241.785,-108.839,171.035,41.816,157.966
C00662=1038.652,241.537,-108.811,171.032,41.815,157.966
C00663=1038.646,241.288,-108.782,171.030,41.814,157.965
C00664=1038.640,241.040,-108.753,171.026,41.812,157.965
C00665=1038.632,240.791,-108.725,171.024,41.811,157.964
C00666=1038.626,240.543,-108.697,171.021,41.810,157.964
C00667=1038.619,240.295,-108.668,171.019,41.808,157.964
C00668=1038.612,240.047,-108.639,171.015,41.807,157.963
C00669=1038.606,239.799,-108.612,171.013,41.806,157.963
C00670=1038.599,239.550,-108.583,171.011,41.805,157.962
C00671=1038.592,239.301,-108.554,171.008,41.803,157.962
C00672=1038.585,239.053,-108.526,171.004,41.802,157.961
C00673=1038.579,238.805,-108.498,171.002,41.801,157.961
C00674=1038.572,238.557,-108.469,170.999,41.799,157.961
C00675=1038.566,238.308,-108.442,170.997,41.798,157.960
C00676=1038.559,238.060,-108.413,170.994,41.797,157.960
C00677=1038.553,237.812,-108.385,170.991,41.795,157.959
C00678=1038.545,237.563,-108.356,170.988,41.794,157.959
C00679=1038.539,237.315,-108.328,170.986,41.793,157.958
C00680=1038.532,237.067,-108.299,170.983,41.792,157.958
C00681=1038.525,236.818,-108.271,170.980,41.790,157.957
C00682=1038.519,236.570,-108.244,170.978,41.789,157.957
C00683=1038.513,236.322,-108.215,170.975,41.788,157.957
C00684=1038.506,236.073,-108.187,170.972,41.786,157.956
C00685=1038.499,235.825,-108.159,170.970,41.785,157.956
C00686=1038.492,235.577,-108.131,170.966,41.784,157.955
C00687=1038.486,235.328,-108.102,170.964,41.783,157.955
C00688=1038.477,235.010,-108.067,170.960,41.781,157.954
C00689=1038.469,234.692,-108.030,170.958,41.779,157.954
C00690=1038.459,234.374,-107.994,170.954,41.778,157.953
C00691=1038.452,234.056,-107.959,170.951,41.776,157.953
C00692=1038.445,233.808,-107.930,170.948,41.775,157.952
C00693=1038.438,233.560,-107.902,170.946,41.774,157.952
C00694=1038.432,233.311,-107.874,170.943,41.772,157.951
C00695=1038.425,233.063,-107.846,170.940,41.771,157.951
C00696=1038.419,232.814,-107.818,170.937,41.770,157.950
C00697=1038.412,232.566,-107.790,170.934,41.768,157.950
C00698=1038.406,232.317,-107.762,170.932,41.767,157.950
C00699=1038.399,232.069,-107.733,170.929,41.766,157.949
C00700=1038.392,231.821,-107.706,170.927,41.765,157.949
C00701=1038.386,231.573,-107.678,170.925,41.763,157.948
C00702=1038.379,231.324,-107.650,170.922,41.762,157.948
C00703=1038.372,231.076,-107.623,170.919,41.761,157.947
C00704=1038.366,230.828,-107.593,170.916,41.759,157.947
C00705=1038.359,230.579,-107.566,170.914,41.758,157.947
C00706=1038.353,230.331,-107.538,170.911,41.757,157.946
C00707=1038.346,230.082,-107.510,170.909,41.756,157.946
C00708=1038.339,229.834,-107.483,170.906,41.754,157.945
C00709=1038.333,229.585,-107.455,170.904,41.753,157.945
C00710=1038.326,229.337,-107.427,170.901,41.752,157.944
C00711=1038.319,229.088,-107.399,170.898,41.751,157.944
C00712=1038.313,228.840,-107.372,170.895,41.749,157.944
C00713=1038.306,228.592,-107.344,170.893,41.748,157.943
C00714=1038.299,228.344,-107.315,170.890,41.747,157.943
C00715=1038.292,228.095,-107.288,170.888,41.746,157.942
C00716=1038.286,227.846,-107.261,170.885,41.744,157.942
C00717=1038.279,227.598,-107.233,170.883,41.743,157.942
C00718=1038.273,227.349,-107.205,170.880,41.742,157.941
C00719=1038.266,227.101,-107.178,170.878,41.740,157.941
C00720=1038.259,226.853,-107.150,170.875,41.740,157.940
C00721=1038.252,226.604,-107.123,170.872,41.738,157.940
C00722=1038.245,226.356,-107.095,170.870,41.737,157.939
C00723=1038.238,226.108,-107.067,170.867,41.736,157.939
C00724=1038.232,225.860,-107.040,170.865,41.735,157.939
C00725=1038.226,225.611,-107.012,170.862,41.734,157.938
C00726=1038.219,225.363,-106.984,170.860,41.732,157.938
C00727=1038.212,225.114,-106.957,170.857,41.731,157.937
C00728=1038.205,224.866,-106.930,170.855,41.729,157.937
C00729=1038.198,224.617,-106.902,170.852,41.728,157.937
C00730=1038.192,224.369,-106.875,170.850,41.727,157.936
C00731=1038.185,224.120,-106.847,170.847,41.726,157.936
C00732=1038.178,223.872,-106.819,170.844,41.724,157.935
C00733=1038.172,223.624,-106.792,170.841,41.724,157.935
C00734=1038.166,223.375,-106.765,170.839,41.723,157.935
C00735=1038.159,223.127,-106.738,170.836,41.721,157.934
C00736=1038.152,222.879,-106.710,170.834,41.720,157.934
C00737=1038.145,222.630,-106.682,170.831,41.718,157.933
C00738=1038.139,222.381,-106.655,170.829,41.717,157.933
C00739=1038.132,222.133,-106.628,170.827,41.716,157.932
C00740=1038.126,221.885,-106.600,170.824,41.715,157.932
C00741=1038.119,221.637,-106.573,170.822,41.713,157.932
C00742=1038.112,221.388,-106.546,170.819,41.712,157.931
C00743=1038.106,221.139,-106.518,170.817,41.711,157.931
C00744=1038.097,220.814,-106.482,170.813,41.709,157.930
C00745=1038.088,220.488,-106.447,170.810,41.708,157.930
C00746=1038.080,220.163,-106.411,170.807,41.706,157.929
C00747=1038.071,219.837,-106.375,170.804,41.705,157.929
C00748=1038.064,219.588,-106.349,170.802,41.703,157.928
C00749=1038.057,219.340,-106.321,170.799,41.702,157.928
C00750=1038.051,219.091,-106.293,170.796,41.701,157.927
C00751=1038.044,218.843,-106.267,170.793,41.700,157.927
C00752=1038.038,218.595,-106.239,170.791,41.699,157.927
C00753=1038.030,218.346,-106.213,170.789,41.698,157.926
C00754=1038.024,218.098,-106.185,170.786,41.696,157.926
C00755=1038.017,217.849,-106.159,170.784,41.695,157.925
C00756=1038.011,217.601,-106.131,170.781,41.694,157.925
C00757=1038.004,217.352,-106.104,170.779,41.693,157.925
C00758=1037.997,217.104,-106.077,170.776,41.692,157.924
C00759=1037.990,216.855,-106.050,170.774,41.690,157.924
C00760=1037.984,216.608,-106.023,170.771,41.689,157.923
C00761=1037.977,216.358,-105.996,170.769,41.688,157.923
C00762=1037.970,216.110,-105.969,170.766,41.686,157.923
C00763=1037.963,215.861,-105.942,170.765,41.685,157.922
C00764=1037.957,215.614,-105.916,170.763,41.684,157.922
C00765=1037.950,215.365,-105.889,170.760,41.683,157.921
C00766=1037.943,215.116,-105.862,170.758,41.682,157.921
C00767=1037.936,214.868,-105.834,170.755,41.680,157.921
C00768=1037.931,214.619,-105.808,170.753,41.679,157.920
C00769=1037.923,214.371,-105.781,170.750,41.678,157.920
C00770=1037.917,214.122,-105.754,170.748,41.677,157.919
C00771=1037.910,213.874,-105.728,170.746,41.676,157.919
C00772=1037.904,213.626,-105.700,170.743,41.675,157.919
C00773=1037.897,213.377,-105.673,170.741,41.673,157.918
C00774=1037.891,213.128,-105.647,170.738,41.672,157.918
C00775=1037.883,212.880,-105.620,170.736,41.671,157.917
C00776=1037.877,212.631,-105.593,170.733,41.670,157.917
C00777=1037.870,212.383,-105.567,170.731,41.669,157.917
C00778=1037.864,212.135,-105.539,170.728,41.667,157.916
C00779=1037.857,211.886,-105.512,170.726,41.666,157.916
C00780=1037.851,211.638,-105.486,170.724,41.664,157.915
C00781=1037.843,211.390,-105.459,170.722,41.663,157.915
C00782=1037.837,211.140,-105.432,170.720,41.662,157.915
C00783=1037.831,210.892,-105.406,170.717,41.661,157.914
C00784=1037.824,210.643,-105.379,170.715,41.660,157.914
C00785=1037.817,210.395,-105.351,170.712,41.659,157.914
C00786=1037.810,210.147,-105.325,170.710,41.657,157.913
C00787=1037.804,209.898,-105.298,170.707,41.656,157.913
C00788=1037.797,209.649,-105.272,170.705,41.655,157.912
C00789=1037.790,209.401,-105.246,170.702,41.654,157.912
C00790=1037.784,209.152,-105.219,170.700,41.653,157.912
C00791=1037.777,208.905,-105.192,170.699,41.652,157.911
C00792=1037.770,208.656,-105.166,170.696,41.650,157.911
C00793=1037.764,208.407,-105.139,170.694,41.649,157.910
C00794=1037.757,208.159,-105.113,170.691,41.648,157.910
C00795=1037.750,207.910,-105.086,170.689,41.646,157.910
C00796=1037.743,207.661,-105.060,170.686,41.645,157.909
C00797=1037.737,207.413,-105.033,170.684,41.644,157.909
C00798=1037.730,207.164,-105.007,170.681,41.643,157.908
C00799=1037.723,206.916,-104.981,170.679,41.642,157.908
C00800=1037.714,206.596,-104.946,170.676,41.640,157.908
C00801=1037.706,206.276,-104.912,170.674,41.639,157.907
C00802=1037.697,205.956,-104.878,170.670,41.637,157.907
C00803=1037.688,205.636,-104.845,170.668,41.636,157.906
C00804=1037.662,204.585,-104.738,170.363,41.532,157.867
C00805=1037.656,204.337,-104.713,170.360,41.531,157.867
C00806=1037.650,204.089,-104.687,170.357,41.531,157.866
C00807=1037.644,203.839,-104.663,170.354,41.530,157.866
C00808=1037.638,203.591,-104.637,170.350,41.530,157.866
C00809=1037.632,203.342,-104.612,170.347,41.529,157.865
C00810=1037.625,203.094,-104.587,170.344,41.529,157.865
C00811=1037.619,202.845,-104.562,170.341,41.529,157.865
C00812=1037.613,202.596,-104.538,170.337,41.528,157.864
C00813=1037.607,202.348,-104.512,170.335,41.528,157.864
C00814=1037.601,202.099,-104.487,170.332,41.527,157.864
C00815=1037.595,201.850,-104.462,170.329,41.527,157.864
C00816=1037.589,201.601,-104.437,170.325,41.526,157.863
C00817=1037.583,201.352,-104.412,170.322,41.526,157.863
C00818=1037.577,201.105,-104.387,170.319,41.526,157.863
C00819=1037.571,200.855,-104.362,170.315,41.525,157.863
C00820=1037.564,200.607,-104.337,170.312,41.525,157.862
C00821=1037.558,200.358,-104.312,170.309,41.524,157.862
C00822=1037.551,200.109,-104.288,170.306,41.524,157.862
C00823=1037.545,199.861,-104.263,170.303,41.524,157.862
C00824=1037.538,199.612,-104.239,170.300,41.524,157.861
C00825=1037.533,199.364,-104.214,170.297,41.523,157.861
C00826=1037.527,199.114,-104.189,170.294,41.523,157.861
C00827=1037.520,198.866,-104.164,170.291,41.523,157.861
C00828=1037.514,198.617,-104.140,170.288,41.523,157.861
C00829=1037.507,198.368,-104.115,170.284,41.522,157.860
C00830=1037.502,198.120,-104.091,170.281,41.522,157.860
C00831=1037.495,197.871,-104.066,170.278,41.521,157.860
C00832=1037.489,197.622,-104.041,170.274,41.521,157.859
C00833=1037.482,197.374,-104.017,170.271,41.521,157.859
C00834=1037.477,197.125,-103.992,170.269,41.521,157.859
C00835=1037.471,196.876,-103.967,170.266,41.520,157.859
C00836=1037.464,196.627,-103.943,170.263,41.520,157.859
C00837=1037.458,196.378,-103.918,170.259,41.520,157.858
C00838=1037.452,196.131,-103.894,170.256,41.520,157.858
C00839=1037.446,195.881,-103.869,170.253,41.519,157.858
C00840=1037.439,195.633,-103.845,170.250,41.519,157.858
C00841=1037.433,195.384,-103.820,170.247,41.519,157.857
C00842=1037.427,195.135,-103.796,170.244,41.519,157.857
C00843=1037.421,194.887,-103.771,170.241,41.518,157.857
C00844=1037.414,194.638,-103.747,170.238,41.518,157.857
C00845=1037.409,194.389,-103.723,170.235,41.518,157.857
C00846=1037.402,194.141,-103.698,170.232,41.518,157.856
C00847=1037.396,193.891,-103.673,170.228,41.517,157.856
C00848=1037.390,193.643,-103.650,170.226,41.517,157.856
C00849=1037.384,193.394,-103.624,170.223,41.517,157.856
C00850=1037.377,193.146,-103.600,170.220,41.517,157.855
C00851=1037.372,192.897,-103.576,170.217,41.516,157.855
C00852=1037.366,192.648,-103.552,170.213,41.516,157.855
C00853=1037.359,192.399,-103.527,170.210,41.516,157.855
C00854=1037.354,192.151,-103.503,170.208,41.516,157.855
C00855=1037.347,191.902,-103.478,170.205,41.515,157.854
C00856=1037.341,191.652,-103.454,170.202,41.515,157.854
C00857=1037.335,191.405,-103.429,170.198,41.515,157.854
C00858=1037.329,191.155,-103.405,170.195,41.515,157.854
C00859=1037.323,190.907,-103.381,170.193,41.514,157.853
C00860=1037.317,190.658,-103.357,170.190,41.514,157.853
C00861=1037.310,190.409,-103.333,170.186,41.514,157.853
C00862=1037.305,190.160,-103.308,170.183,41.514,157.853
C00863=1037.298,189.912,-103.284,170.181,41.513,157.852
C00864=1037.293,189.663,-103.259,170.178,41.513,157.852
C00865=1037.286,189.379,-103.232,170.175,41.513,157.852
C00866=1037.279,189.095,-103.204,170.170,41.513,157.852
C00867=1037.272,188.810,-103.177,170.167,41.512,157.852
C00868=1037.265,188.526,-103.149,170.164,41.512,157.851
C00869=1037.258,188.278,-103.125,170.161,41.512,157.851
C00870=1037.253,188.028,-103.101,170.159,41.512,157.851
C00871=1037.247,187.780,-103.077,170.155,41.511,157.851
C00872=1037.241,187.531,-103.052,170.152,41.511,157.850
C00873=1037.235,187.283,-103.029,170.149,41.511,157.850
C00874=1037.229,187.033,-103.004,170.147,41.510,157.850
C00875=1037.223,186.785,-102.980,170.144,41.510,157.850
C00876=1037.217,186.536,-102.956,170.140,41.510,157.849
C00877=1037.211,186.287,-102.932,170.137,41.510,157.849
C00878=1037.205,186.038,-102.907,170.135,41.509,157.849
C00879=1037.199,185.790,-102.884,170.132,41.510,157.849
C00880=1037.193,185.541,-102.859,170.129,41.510,157.849
C00881=1037.187,185.292,-102.835,170.127,41.509,157.849
C00882=1037.182,185.044,-102.811,170.123,41.509,157.848
C00883=1037.175,184.795,-102.787,170.120,41.509,157.848
C00884=1037.169,184.546,-102.763,170.117,41.508,157.848
C00885=1037.163,184.297,-102.739,170.115,41.508,157.848
C00886=1037.157,184.049,-102.715,170.111,41.508,157.847
C00887=1037.152,183.800,-102.691,170.108,41.508,157.847
C00888=1037.145,183.551,-102.667,170.106,41.507,157.847
C00889=1037.140,183.302,-102.643,170.103,41.508,157.847
C00890=1037.133,183.053,-102.619,170.100,41.507,157.847
C00891=1037.127,182.805,-102.596,170.097,41.507,157.846
C00892=1037.120,182.556,-102.573,170.095,41.507,157.846
C00893=1037.114,182.307,-102.549,170.091,41.507,157.846
C00894=1037.108,182.058,-102.525,170.088,41.508,157.846
C00895=1037.102,181.809,-102.502,170.085,41.507,157.846
C00896=1037.095,181.560,-102.478,170.083,41.508,157.846
C00897=1037.089,181.312,-102.455,170.080,41.507,157.845
C00898=1037.083,181.063,-102.431,170.077,41.507,157.845
C00899=1037.077,180.814,-102.408,170.074,41.508,157.845
C00900=1037.070,180.565,-102.384,170.071,41.507,157.845
C00901=1037.064,180.317,-102.361,170.068,41.508,157.845
C00902=1037.057,180.068,-102.337,170.065,41.507,157.845
C00903=1037.051,179.819,-102.314,170.062,41.508,157.845
C00904=1037.045,179.570,-102.290,170.060,41.507,157.844
C00905=1037.039,179.321,-102.267,170.057,41.507,157.844
C00906=1037.033,179.073,-102.244,170.054,41.508,157.844
C00907=1037.027,178.823,-102.220,170.052,41.507,157.844
C00908=1037.021,178.575,-102.197,170.049,41.508,157.844
C00909=1037.013,178.326,-102.174,170.045,41.507,157.843
C00910=1037.007,178.077,-102.150,170.042,41.508,157.843
C00911=1037.001,177.828,-102.127,170.040,41.507,157.843
C00912=1036.995,177.579,-102.103,170.037,41.508,157.843
C00913=1036.989,177.330,-102.080,170.034,41.508,157.843
C00914=1036.983,177.082,-102.056,170.032,41.507,157.843
C00915=1036.977,176.833,-102.033,170.029,41.508,157.843
C00916=1036.970,176.585,-102.010,170.025,41.507,157.842
C00917=1036.964,176.335,-101.987,170.023,41.508,157.842
C00918=1036.958,176.087,-101.963,170.020,41.507,157.842
C00919=1036.952,175.838,-101.940,170.017,41.508,157.842
C00920=1036.946,175.588,-101.917,170.014,41.508,157.842
C00921=1036.940,175.340,-101.893,170.012,41.508,157.842
C00922=1036.934,175.091,-101.871,170.009,41.508,157.841
C00923=1036.927,174.842,-101.847,170.006,41.508,157.841
C00924=1036.921,174.594,-101.824,170.003,41.508,157.841
C00925=1036.915,174.345,-101.801,170.000,41.508,157.841
C00926=1036.909,174.096,-101.777,169.997,41.508,157.841
C00927=1036.903,173.847,-101.754,169.995,41.508,157.841
C00928=1036.897,173.598,-101.731,169.992,41.508,157.841
C00929=1036.889,173.313,-101.705,169.989,41.508,157.840
C00930=1036.883,173.029,-101.678,169.986,41.508,157.840
C00931=1036.875,172.744,-101.652,169.982,41.508,157.840
C00932=1036.869,172.460,-101.625,169.979,41.508,157.840
C00933=1036.862,172.211,-101.602,169.976,41.508,157.840
C00934=1036.856,171.962,-101.579,169.974,41.508,157.840
C00935=1036.850,171.713,-101.556,169.971,41.508,157.839
C00936=1036.844,171.465,-101.532,169.969,41.508,157.839
C00937=1036.839,171.216,-101.509,169.966,41.508,157.839
C00938=1036.832,170.966,-101.486,169.963,41.508,157.839
C00939=1036.826,170.717,-101.464,169.961,41.508,157.839
C00940=1036.820,170.469,-101.440,169.958,41.508,157.839
C00941=1036.814,170.220,-101.417,169.955,41.508,157.838
C00942=1036.808,169.971,-101.394,169.952,41.508,157.838
C00943=1036.802,169.722,-101.371,169.949,41.508,157.838
C00944=1036.795,169.473,-101.348,169.947,41.508,157.838
C00945=1036.790,169.224,-101.325,169.944,41.508,157.838
C00946=1036.784,168.976,-101.302,169.942,41.508,157.838
C00947=1036.778,168.727,-101.279,169.939,41.508,157.838
C00948=1036.772,168.478,-101.256,169.936,41.509,157.837
C00949=1036.765,168.229,-101.233,169.933,41.508,157.837
C00950=1036.759,167.980,-101.210,169.930,41.509,157.837
C00951=1036.754,167.731,-101.187,169.928,41.508,157.837
C00952=1036.748,167.482,-101.164,169.925,41.509,157.837
C00953=1036.742,167.234,-101.141,169.923,41.508,157.837
C00954=1036.736,166.984,-101.117,169.920,41.509,157.837
C00955=1036.729,166.736,-101.095,169.917,41.508,157.836
C00956=1036.723,166.487,-101.072,169.915,41.509,157.836
C00957=1036.718,166.238,-101.049,169.911,41.508,157.836
C00958=1036.712,165.989,-101.026,169.909,41.509,157.836
C00959=1036.705,165.741,-101.004,169.906,41.509,157.836
C00960=1036.700,165.492,-100.981,169.904,41.509,157.836
C00961=1036.694,165.243,-100.958,169.901,41.509,157.836
C00962=1036.688,164.994,-100.935,169.899,41.509,157.835
C00963=1036.683,164.745,-100.912,169.896,41.509,157.835
C00964=1036.676,164.496,-100.889,169.893,41.509,157.835
C00965=1036.670,164.247,-100.866,169.891,41.509,157.835
C00966=1036.664,163.998,-100.843,169.887,41.509,157.835
C00967=1036.658,163.749,-100.821,169.885,41.509,157.835
C00968=1036.653,163.500,-100.798,169.882,41.509,157.834
C00969=1036.646,163.251,-100.775,169.880,41.509,157.834
C00970=1036.640,163.003,-100.752,169.877,41.509,157.834
C00971=1036.635,162.754,-100.729,169.875,41.509,157.834
C00972=1036.629,162.505,-100.706,169.872,41.509,157.834
C00973=1036.622,162.256,-100.684,169.870,41.509,157.834
C00974=1036.617,162.007,-100.661,169.867,41.509,157.834
C00975=1036.611,161.758,-100.639,169.864,41.509,157.833
C00976=1036.606,161.509,-100.616,169.861,41.510,157.833
C00977=1036.599,161.260,-100.594,169.859,41.509,157.833
C00978=1036.593,161.011,-100.571,169.856,41.510,157.833
C00979=1036.588,160.763,-100.548,169.854,41.509,157.833
C00980=1036.582,160.514,-100.525,169.851,41.510,157.833
C00981=1036.576,160.265,-100.502,169.849,41.509,157.833
C00982=1036.570,160.016,-100.480,169.846,41.510,157.833
C00983=1036.564,159.767,-100.457,169.844,41.510,157.832
C00984=1036.558,159.518,-100.435,169.841,41.510,157.832
C00985=1036.551,159.269,-100.412,169.839,41.510,157.832
C00986=1036.546,159.020,-100.390,169.835,41.510,157.832
C00987=1036.539,158.771,-100.368,169.833,41.511,157.832
C00988=1036.534,158.522,-100.345,169.830,41.510,157.832
C00989=1036.528,158.273,-100.323,169.828,41.511,157.832
C00990=1036.521,158.025,-100.301,169.825,41.511,157.832
C00991=1036.515,157.776,-100.278,169.823,41.511,157.832
C00992=1036.509,157.527,-100.256,169.820,41.511,157.831
C00993=1036.502,157.241,-100.230,169.817,41.512,157.831
C00994=1036.495,156.956,-100.205,169.814,41.512,157.831
C00995=1036.488,156.671,-100.179,169.811,41.512,157.831
C00996=1036.481,156.386,-100.154,169.809,41.512,157.831
C00997=1036.475,156.137,-100.132,169.806,41.512,157.831
C00998=1036.469,155.888,-100.110,169.803,41.513,157.831
C00999=1036.463,155.639,-100.087,169.801,41.513,157.831
C01000=1036.456,155.391,-100.065,169.797,41.513,157.830
C01001=1036.451,155.141,-100.043,169.795,41.513,157.830
C01002=1036.444,154.893,-100.021,169.793,41.513,157.830
C01003=1036.438,154.643,-99.999,169.790,41.514,157.830
C01004=1036.432,154.395,-99.976,169.788,41.513,157.830
C01005=1036.426,154.145,-99.954,169.785,41.514,157.830
C01006=1036.420,153.897,-99.932,169.783,41.514,157.830
C01007=1036.414,153.648,-99.910,169.780,41.514,157.830
C01008=1036.408,153.399,-99.887,169.778,41.515,157.830
C01009=1036.402,153.149,-99.866,169.775,41.515,157.829
C01010=1036.396,152.900,-99.844,169.773,41.515,157.829
C01011=1036.390,152.652,-99.822,169.770,41.515,157.829
C01012=1036.384,152.403,-99.800,169.768,41.515,157.829
C01013=1036.378,152.154,-99.778,169.765,41.516,157.829
C01014=1036.372,151.905,-99.756,169.763,41.516,157.829
C01015=1036.365,151.657,-99.734,169.760,41.516,157.829
C01016=1036.359,151.407,-99.712,169.758,41.517,157.829
C01017=1036.353,151.158,-99.690,169.754,41.516,157.829
C01018=1036.346,150.910,-99.668,169.752,41.517,157.829
C01019=1036.341,150.660,-99.646,169.749,41.517,157.828
C01020=1036.335,150.411,-99.624,169.747,41.517,157.828
C01021=1036.329,150.163,-99.602,169.744,41.518,157.828
C01022=1036.323,149.914,-99.580,169.742,41.518,157.828
C01023=1036.317,149.664,-99.559,169.739,41.518,157.828
C01024=1036.310,149.416,-99.536,169.737,41.518,157.828
C01025=1036.305,149.166,-99.514,169.735,41.518,157.828
C01026=1036.299,148.917,-99.493,169.732,41.519,157.828
C01027=1036.292,148.669,-99.470,169.730,41.519,157.828
C01028=1036.286,148.419,-99.449,169.727,41.519,157.828
C01029=1036.280,148.171,-99.427,169.725,41.520,157.828
C01030=1036.274,147.922,-99.406,169.722,41.520,157.827
C01031=1036.268,147.673,-99.383,169.720,41.520,157.827
C01032=1036.262,147.424,-99.362,169.716,41.520,157.827
C01033=1036.255,147.175,-99.340,169.714,41.520,157.827
C01034=1036.250,146.925,-99.318,169.711,41.521,157.827
C01035=1036.244,146.677,-99.297,169.709,41.521,157.827
C01036=1036.237,146.428,-99.275,169.707,41.521,157.827
C01037=1036.231,146.179,-99.253,169.704,41.522,157.827
C01038=1036.225,145.930,-99.232,169.702,41.522,157.827
C01039=1036.219,145.681,-99.210,169.699,41.522,157.827
C01040=1036.213,145.432,-99.188,169.697,41.523,157.827
C01041=1036.206,145.182,-99.167,169.694,41.523,157.826
C01042=1036.201,144.934,-99.145,169.692,41.523,157.826
C01043=1036.195,144.685,-99.124,169.689,41.524,157.826
C01044=1036.188,144.436,-99.101,169.687,41.524,157.826
C01045=1036.182,144.187,-99.080,169.685,41.524,157.826
C01046=1036.176,143.938,-99.058,169.682,41.525,157.826
C01047=1036.170,143.689,-99.037,169.680,41.525,157.826
C01048=1036.163,143.440,-99.016,169.677,41.525,157.826
C01049=1036.157,143.191,-98.994,169.675,41.525,157.826
C01050=1036.151,142.942,-98.973,169.672,41.526,157.826
C01051=1036.146,142.693,-98.951,169.670,41.526,157.826
C01052=1036.139,142.444,-98.930,169.668,41.526,157.826
C01053=1036.133,142.195,-98.908,169.665,41.527,157.825
C01054=1036.127,141.946,-98.886,169.663,41.526,157.825
C01055=1036.121,141.697,-98.865,169.660,41.527,157.825
C01056=1036.115,141.448,-98.843,169.658,41.527,157.825
C01057=1036.107,141.163,-98.819,169.655,41.527,157.825
C01058=1036.101,140.877,-98.794,169.652,41.528,157.825
C01059=1036.095,140.592,-98.769,169.650,41.528,157.825
C01060=1036.087,140.306,-98.745,169.646,41.529,157.825
C01061=1036.081,140.058,-98.723,169.643,41.529,157.825
C01062=1036.075,139.808,-98.703,169.641,41.529,157.825
C01063=1036.069,139.559,-98.681,169.639,41.529,157.825
C01064=1036.064,139.310,-98.660,169.636,41.530,157.824
C01065=1036.057,139.061,-98.639,169.634,41.530,157.824
C01066=1036.050,138.812,-98.617,169.631,41.530,157.824
C01067=1036.044,138.563,-98.595,169.629,41.531,157.824
C01068=1036.039,138.314,-98.574,169.627,41.531,157.824
C01069=1036.032,138.066,-98.553,169.624,41.531,157.824
C01070=1036.026,137.816,-98.532,169.622,41.532,157.824
C01071=1036.020,137.567,-98.511,169.619,41.532,157.824
C01072=1036.014,137.318,-98.489,169.617,41.532,157.824
C01073=1036.007,137.069,-98.468,169.615,41.533,157.824
C01074=1036.002,136.821,-98.447,169.612,41.534,157.824
C01075=1035.996,136.571,-98.426,169.610,41.534,157.824
C01076=1035.989,136.322,-98.405,169.607,41.534,157.824
C01077=1035.983,136.073,-98.383,169.605,41.535,157.824
C01078=1035.977,135.824,-98.362,169.603,41.535,157.824
C01079=1035.971,135.575,-98.342,169.600,41.535,157.823
C01080=1035.965,135.325,-98.320,169.598,41.536,157.823
C01081=1035.959,135.077,-98.299,169.595,41.536,157.823
C01082=1035.952,134.828,-98.278,169.593,41.536,157.823
C01083=1035.946,134.578,-98.257,169.591,41.536,157.823
C01084=1035.941,134.330,-98.236,169.588,41.537,157.823
C01085=1035.934,134.081,-98.215,169.586,41.537,157.823
C01086=1035.928,133.832,-98.194,169.584,41.537,157.823
C01087=1035.922,133.582,-98.172,169.581,41.538,157.823
C01088=1035.915,133.334,-98.151,169.579,41.539,157.823
C01089=1035.910,133.084,-98.131,169.576,41.539,157.823
C01090=1035.903,132.836,-98.110,169.574,41.539,157.823
C01091=1035.897,132.586,-98.088,169.572,41.540,157.823
C01092=1035.892,132.337,-98.068,169.569,41.540,157.823
C01093=1035.885,132.088,-98.046,169.567,41.540,157.822
C01094=1035.879,131.840,-98.025,169.565,41.541,157.822
C01095=1035.874,131.590,-98.004,169.562,41.541,157.822
C01096=1035.867,131.341,-97.983,169.560,41.541,157.822
C01097=1035.861,131.092,-97.963,169.558,41.541,157.822
C01098=1035.854,130.843,-97.942,169.555,41.542,157.822
C01099=1035.849,130.594,-97.921,169.553,41.542,157.822
C01100=1035.842,130.345,-97.900,169.550,41.543,157.822
C01101=1035.836,130.096,-97.880,169.548,41.543,157.822
C01102=1035.830,129.847,-97.858,169.546,41.544,157.822
C01103=1035.824,129.598,-97.838,169.543,41.544,157.822
C01104=1035.817,129.349,-97.817,169.541,41.545,157.822
C01105=1035.811,129.100,-97.797,169.538,41.545,157.822
C01106=1035.805,128.851,-97.776,169.536,41.546,157.822
C01107=1035.799,128.602,-97.756,169.534,41.546,157.822
C01108=1035.792,128.353,-97.734,169.531,41.547,157.822
C01109=1035.786,128.103,-97.714,169.529,41.547,157.822
C01110=1035.780,127.854,-97.694,169.527,41.547,157.822
C01111=1035.774,127.605,-97.672,169.524,41.548,157.821
C01112=1035.768,127.356,-97.652,169.522,41.548,157.821
C01113=1035.761,127.107,-97.631,169.519,41.549,157.821
C01114=1035.755,126.859,-97.611,169.517,41.549,157.821
C01115=1035.749,126.609,-97.590,169.515,41.550,157.821
C01116=1035.742,126.360,-97.569,169.512,41.550,157.821
C01117=1035.736,126.111,-97.549,169.510,41.550,157.821
C01118=1035.730,125.861,-97.528,169.508,41.551,157.821
C01119=1035.724,125.613,-97.508,169.505,41.552,157.821
C01120=1035.717,125.364,-97.487,169.503,41.552,157.821
C01121=1035.710,125.078,-97.464,169.500,41.552,157.821
C01122=1035.703,124.793,-97.440,169.498,41.553,157.821
C01123=1035.696,124.507,-97.416,169.495,41.554,157.821
C01124=1035.689,124.222,-97.393,169.492,41.554,157.821
C01125=1035.683,123.972,-97.372,169.490,41.554,157.821
C01126=1035.677,123.723,-97.352,169.487,41.555,157.821
C01127=1035.671,123.474,-97.331,169.485,41.556,157.821
C01128=1035.664,123.226,-97.311,169.483,41.556,157.821
C01129=1035.658,122.976,-97.290,169.480,41.556,157.821
C01130=1035.653,122.727,-97.270,169.478,41.557,157.821
C01131=1035.646,122.477,-97.249,169.476,41.557,157.820
C01132=1035.640,122.229,-97.229,169.473,41.558,157.820
C01133=1035.634,121.979,-97.208,169.471,41.558,157.820
C01134=1035.628,121.731,-97.188,169.469,41.558,157.820
C01135=1035.621,121.481,-97.168,169.466,41.559,157.820
C01136=1035.615,121.233,-97.147,169.464,41.559,157.820
C01137=1035.609,120.983,-97.126,169.462,41.560,157.820
C01138=1035.603,120.734,-97.106,169.460,41.560,157.820
C01139=1035.597,120.485,-97.086,169.457,41.561,157.820
C01140=1035.591,120.236,-97.066,169.455,41.561,157.820
C01141=1035.585,119.987,-97.045,169.453,41.561,157.820
C01142=1035.578,119.738,-97.024,169.450,41.562,157.820
C01143=1035.572,119.489,-97.004,169.448,41.562,157.820
C01144=1035.566,119.239,-96.983,169.446,41.563,157.820
C01145=1035.561,118.990,-96.963,169.443,41.563,157.820
C01146=1035.555,118.742,-96.943,169.441,41.563,157.820
C01147=1035.548,118.492,-96.923,169.439,41.564,157.820
C01148=1035.543,118.243,-96.903,169.436,41.565,157.820
C01149=1035.536,117.994,-96.881,169.434,41.565,157.820
C01150=1035.530,117.745,-96.862,169.432,41.565,157.820
C01151=1035.524,117.497,-96.842,169.430,41.566,157.819
C01152=1035.518,117.247,-96.821,169.427,41.566,157.819
C01153=1035.512,116.998,-96.801,169.425,41.566,157.819
C01154=1035.506,116.749,-96.781,169.423,41.567,157.819
C01155=1035.499,116.500,-96.760,169.420,41.568,157.819
C01156=1035.494,116.250,-96.740,169.418,41.568,157.819
C01157=1035.488,116.002,-96.720,169.416,41.568,157.819
C01158=1035.481,115.752,-96.700,169.414,41.568,157.819
C01159=1035.475,115.503,-96.680,169.411,41.569,157.819
C01160=1035.470,115.254,-96.659,169.409,41.570,157.819
C01161=1035.464,115.005,-96.639,169.407,41.570,157.819
C01162=1035.458,114.756,-96.619,169.405,41.570,157.819
C01163=1035.452,114.507,-96.599,169.402,41.571,157.819
C01164=1035.446,114.257,-96.578,169.400,41.571,157.819
C01165=1035.440,114.008,-96.558,169.398,41.571,157.819
C01166=1035.434,113.760,-96.538,169.396,41.571,157.819
C01167=1035.427,113.510,-96.518,169.393,41.572,157.819
C01168=1035.422,113.261,-96.497,169.391,41.573,157.819
C01169=1035.415,113.012,-96.478,169.389,41.573,157.819
C01170=1035.409,112.763,-96.457,169.386,41.573,157.818
C01171=1035.403,112.514,-96.437,169.384,41.574,157.818
C01172=1035.396,112.265,-96.417,169.382,41.574,157.818
C01173=1035.390,112.016,-96.397,169.379,41.575,157.818
C01174=1035.384,111.766,-96.378,169.377,41.575,157.818
C01175=1035.378,111.518,-96.358,169.375,41.576,157.818
C01176=1035.372,111.268,-96.338,169.373,41.576,157.818
C01177=1035.366,111.019,-96.318,169.370,41.577,157.818
C01178=1035.360,110.770,-96.298,169.368,41.578,157.818
C01179=1035.353,110.520,-96.278,169.366,41.578,157.818
C01180=1035.347,110.271,-96.258,169.363,41.578,157.818
C01181=1035.342,110.023,-96.238,169.361,41.579,157.818
C01182=1035.335,109.773,-96.218,169.359,41.579,157.818
C01183=1035.329,109.524,-96.198,169.357,41.580,157.818
C01184=1035.322,109.275,-96.179,169.354,41.581,157.818
C01185=1035.316,108.989,-96.156,169.352,41.581,157.818
C01186=1035.308,108.703,-96.134,169.349,41.581,157.818
C01187=1035.301,108.418,-96.110,169.347,41.583,157.818
C01188=1035.294,108.132,-96.088,169.344,41.583,157.818
C01189=1035.288,107.882,-96.068,169.342,41.584,157.818
C01190=1035.282,107.633,-96.048,169.340,41.584,157.818
C01191=1035.275,107.385,-96.029,169.338,41.584,157.818
C01192=1035.269,107.135,-96.010,169.336,41.585,157.818
C01193=1035.263,106.886,-95.989,169.333,41.586,157.818
C01194=1035.257,106.637,-95.969,169.331,41.586,157.818
C01195=1035.251,106.388,-95.950,169.329,41.587,157.818
C01196=1035.244,106.139,-95.931,169.326,41.587,157.818
C01197=1035.238,105.890,-95.911,169.324,41.588,157.818
C01198=1035.232,105.640,-95.891,169.322,41.588,157.818
C01199=1035.226,105.391,-95.871,169.320,41.589,157.818
C01200=1035.220,105.142,-95.852,169.317,41.589,157.817
C01201=1035.213,104.893,-95.832,169.315,41.590,157.818
C01202=1035.207,104.644,-95.812,169.313,41.590,157.817
C01203=1035.201,104.395,-95.793,169.310,41.591,157.817
C01204=1035.195,104.146,-95.773,169.308,41.592,157.817
C01205=1035.188,103.896,-95.754,169.306,41.592,157.817
C01206=1035.182,103.647,-95.734,169.304,41.592,157.817
C01207=1035.176,103.398,-95.714,169.301,41.593,157.817
C01208=1035.171,103.149,-95.695,169.299,41.593,157.817
C01209=1035.165,102.900,-95.675,169.297,41.594,157.817
C01210=1035.157,102.650,-95.656,169.295,41.594,157.817
C01211=1035.151,102.401,-95.636,169.292,41.595,157.817
C01212=1035.146,102.152,-95.617,169.290,41.595,157.817
C01213=1035.140,101.903,-95.597,169.288,41.596,157.817
C01214=1035.133,101.654,-95.578,169.286,41.596,157.817
C01215=1035.127,101.405,-95.558,169.283,41.597,157.817
C01216=1035.121,101.155,-95.539,169.281,41.597,157.817
C01217=1035.115,100.906,-95.519,169.279,41.598,157.817
C01218=1035.109,100.657,-95.500,169.277,41.598,157.817
C01219=1035.103,100.408,-95.480,169.274,41.599,157.817
C01220=1035.097,100.159,-95.461,169.272,41.599,157.817
C01221=1035.091,99.910,-95.441,169.270,41.600,157.817
C01222=1035.085,99.661,-95.422,169.268,41.600,157.817
C01223=1035.078,99.411,-95.403,169.266,41.601,157.817
C01224=1035.072,99.162,-95.383,169.264,41.601,157.817
C01225=1035.066,98.913,-95.364,169.262,41.602,157.817
C01226=1035.059,98.664,-95.345,169.259,41.603,157.817
C01227=1035.053,98.415,-95.325,169.257,41.603,157.817
C01228=1035.046,98.165,-95.306,169.255,41.604,157.817
C01229=1035.041,97.916,-95.287,169.253,41.604,157.817
C01230=1035.034,97.667,-95.268,169.250,41.605,157.817
C01231=1035.028,97.418,-95.249,169.248,41.606,157.817
C01232=1035.022,97.169,-95.230,169.246,41.606,157.817
C01233=1035.016,96.920,-95.210,169.243,41.607,157.817
C01234=1035.009,96.671,-95.191,169.241,41.607,157.816
C01235=1035.004,96.421,-95.172,169.239,41.608,157.817
C01236=1034.996,96.172,-95.152,169.237,41.608,157.816
C01237=1034.991,95.923,-95.133,169.234,41.609,157.817
C01238=1034.984,95.674,-95.114,169.232,41.610,157.816
C01239=1034.979,95.424,-95.095,169.230,41.610,157.816
C01240=1034.972,95.176,-95.076,169.228,41.611,157.816
C01241=1034.965,94.926,-95.057,169.225,41.611,157.816
C01242=1034.960,94.677,-95.038,169.223,41.612,157.816
C01243=1034.953,94.428,-95.019,169.221,41.612,157.816
C01244=1034.947,94.179,-94.999,169.219,41.613,157.816
C01245=1034.941,93.930,-94.981,169.216,41.614,157.816
C01246=1034.935,93.680,-94.961,169.214,41.614,157.816
C01247=1034.928,93.431,-94.942,169.212,41.614,157.816
C01248=1034.923,93.181,-94.923,169.211,41.615,157.816
C01249=1034.916,92.896,-94.901,169.208,41.616,157.816
C01250=1034.909,92.610,-94.880,169.205,41.617,157.816
C01251=1034.901,92.324,-94.857,169.203,41.617,157.816
C01252=1034.895,92.039,-94.836,169.200,41.618,157.816
C01253=1034.888,91.790,-94.817,169.198,41.618,157.816
C01254=1034.882,91.541,-94.797,169.196,41.618,157.816
C01255=1034.876,91.292,-94.779,169.194,41.619,157.816
C01256=1034.870,91.042,-94.759,169.191,41.620,157.816
C01257=1034.864,90.793,-94.741,169.189,41.620,157.816
C01258=1034.858,90.544,-94.722,169.187,41.621,157.816
C01259=1034.852,90.294,-94.703,169.185,41.621,157.816
C01260=1034.846,90.045,-94.684,169.182,41.622,157.816
C01261=1034.839,89.797,-94.664,169.180,41.623,157.816
C01262=1034.832,89.547,-94.645,169.178,41.623,157.816
C01263=1034.826,89.298,-94.627,169.176,41.624,157.816
C01264=1034.820,89.048,-94.607,169.173,41.624,157.816
C01265=1034.814,88.799,-94.589,169.171,41.625,157.816
C01266=1034.807,88.550,-94.570,169.169,41.625,157.816
C01267=1034.801,88.301,-94.551,169.166,41.626,157.816
C01268=1034.795,88.051,-94.534,169.164,41.627,157.816
C01269=1034.788,87.802,-94.515,169.162,41.628,157.816
C01270=1034.782,87.553,-94.496,169.160,41.628,157.816
C01271=1034.776,87.303,-94.477,169.158,41.629,157.816
C01272=1034.770,87.054,-94.458,169.156,41.629,157.816
C01273=1034.763,86.805,-94.440,169.154,41.630,157.816
C01274=1034.757,86.556,-94.421,169.152,41.630,157.816
C01275=1034.751,86.307,-94.402,169.149,41.631,157.816
C01276=1034.745,86.057,-94.383,169.147,41.632,157.816
C01277=1034.738,85.808,-94.365,169.145,41.633,157.816
C01278=1034.732,85.559,-94.346,169.142,41.633,157.816
C01279=1034.725,85.310,-94.327,169.140,41.634,157.816
C01280=1034.719,85.061,-94.309,169.138,41.634,157.816
C01281=1034.714,84.811,-94.290,169.136,41.635,157.816
C01282=1034.707,84.562,-94.271,169.133,41.635,157.816
C01283=1034.701,84.313,-94.253,169.131,41.636,157.816
C01284=1034.694,84.064,-94.234,169.129,41.637,157.816
C01285=1034.688,83.815,-94.216,169.127,41.638,157.816
C01286=1034.682,83.566,-94.197,169.124,41.638,157.816
C01287=1034.676,83.317,-94.178,169.122,41.639,157.816
C01288=1034.670,83.067,-94.160,169.120,41.639,157.816
C01289=1034.664,82.818,-94.141,169.118,41.639,157.815
C01290=1034.657,82.569,-94.123,169.116,41.640,157.815
C01291=1034.651,82.319,-94.104,169.114,41.641,157.815
C01292=1034.645,82.070,-94.085,169.112,41.642,157.815
C01293=1034.639,81.821,-94.066,169.110,41.642,157.815
C01294=1034.633,81.571,-94.048,169.107,41.643,157.815
C01295=1034.626,81.322,-94.030,169.105,41.643,157.815
C01296=1034.620,81.073,-94.011,169.103,41.644,157.815
C01297=1034.614,80.825,-93.993,169.101,41.644,157.815
C01298=1034.608,80.575,-93.975,169.099,41.645,157.815
C01299=1034.601,80.326,-93.956,169.096,41.646,157.815
C01300=1034.596,80.076,-93.937,169.094,41.646,157.815
C01301=1034.589,79.827,-93.918,169.092,41.647,157.815
C01302=1034.583,79.577,-93.900,169.090,41.647,157.815
C01303=1034.577,79.328,-93.882,169.087,41.648,157.815
C01304=1034.570,79.079,-93.863,169.085,41.649,157.815
C01305=1034.565,78.831,-93.845,169.083,41.649,157.815
C01306=1034.558,78.581,-93.827,169.081,41.650,157.815
C01307=1034.553,78.332,-93.807,169.078,41.650,157.815
C01308=1034.546,78.082,-93.789,169.076,41.651,157.815
C01309=1034.540,77.833,-93.771,169.074,41.651,157.815
C01310=1034.534,77.584,-93.752,169.073,41.652,157.815
C01311=1034.528,77.334,-93.734,169.069,41.653,157.815
C01312=1034.521,77.085,-93.716,169.068,41.654,157.815
C01313=1034.514,76.799,-93.695,169.066,41.654,157.815
C01314=1034.507,76.514,-93.674,169.063,41.655,157.815
C01315=1034.500,76.228,-93.653,169.060,41.655,157.815
C01316=1034.493,75.942,-93.633,169.058,41.656,157.815
C01317=1034.486,75.693,-93.614,169.056,41.656,157.815
C01318=1034.480,75.444,-93.595,169.053,41.658,157.815
C01319=1034.474,75.194,-93.578,169.051,41.658,157.815
C01320=1034.467,74.945,-93.559,169.049,41.659,157.815
C01321=1034.462,74.696,-93.541,169.046,41.660,157.815
C01322=1034.455,74.447,-93.523,169.044,41.660,157.815
C01323=1034.448,74.197,-93.505,169.042,41.661,157.815
C01324=1034.442,73.948,-93.487,169.040,41.661,157.815
C01325=1034.436,73.698,-93.469,169.037,41.662,157.815
C01326=1034.429,73.449,-93.450,169.035,41.663,157.815
C01327=1034.424,73.200,-93.433,169.034,41.663,157.815
C01328=1034.417,72.951,-93.414,169.032,41.664,157.815
C01329=1034.411,72.702,-93.397,169.029,41.665,157.815
C01330=1034.404,72.452,-93.378,169.027,41.665,157.815
C01331=1034.399,72.203,-93.360,169.025,41.666,157.815
C01332=1034.393,71.954,-93.342,169.023,41.666,157.815
C01333=1034.386,71.705,-93.324,169.020,41.667,157.815
C01334=1034.380,71.455,-93.306,169.018,41.668,157.815
C01335=1034.374,71.206,-93.287,169.016,41.668,157.815
C01336=1034.367,70.957,-93.270,169.014,41.669,157.815
C01337=1034.361,70.708,-93.252,169.011,41.670,157.815
C01338=1034.355,70.458,-93.234,169.009,41.670,157.815
C01339=1034.349,70.208,-93.216,169.007,41.671,157.815
C01340=1034.343,69.960,-93.197,169.005,41.671,157.815
C01341=1034.337,69.710,-93.179,169.002,41.672,157.815
C01342=1034.330,69.461,-93.162,169.000,41.673,157.815
C01343=1034.323,69.212,-93.143,168.998,41.674,157.815
C01344=1034.318,68.963,-93.126,168.996,41.674,157.815
C01345=1034.312,68.713,-93.108,168.994,41.675,157.815
C01346=1034.305,68.464,-93.090,168.992,41.675,157.815
C01347=1034.299,68.214,-93.072,168.990,41.676,157.815
C01348=1034.293,67.965,-93.054,168.988,41.677,157.815
C01349=1034.286,67.716,-93.036,168.985,41.677,157.815
C01350=1034.280,67.467,-93.018,168.983,41.678,157.815
C01351=1034.274,67.217,-93.001,168.981,41.679,157.815
C01352=1034.267,66.968,-92.984,168.979,41.679,157.815
C01353=1034.261,66.719,-92.965,168.976,41.680,157.815
C01354=1034.255,66.469,-92.947,168.974,41.681,157.815
C01355=1034.249,66.221,-92.930,168.972,41.681,157.815
C01356=1034.242,65.971,-92.912,168.969,41.682,157.815
C01357=1034.236,65.722,-92.893,168.967,41.683,157.815
C01358=1034.229,65.472,-92.876,168.965,41.683,157.815
C01359=1034.224,65.223,-92.858,168.964,41.684,157.815
C01360=1034.218,64.974,-92.841,168.961,41.685,157.815
C01361=1034.211,64.724,-92.823,168.959,41.686,157.815
C01362=1034.205,64.476,-92.805,168.957,41.686,157.815
C01363=1034.198,64.226,-92.788,168.955,41.687,157.815
C01364=1034.192,63.977,-92.770,168.952,41.687,157.815
C01365=1034.186,63.727,-92.752,168.950,41.688,157.815
C01366=1034.179,63.478,-92.735,168.948,41.689,157.815
C01367=1034.173,63.228,-92.717,168.946,41.689,157.815
C01368=1034.166,62.979,-92.699,168.943,41.690,157.815
C01369=1034.160,62.730,-92.683,168.941,41.691,157.815
C01370=1034.154,62.480,-92.665,168.939,41.692,157.815
C01371=1034.147,62.231,-92.647,168.936,41.693,157.815
C01372=1034.141,61.982,-92.630,168.935,41.694,157.815
C01373=1034.135,61.733,-92.612,168.933,41.694,157.815
C01374=1034.128,61.484,-92.594,168.930,41.695,157.815
C01375=1034.121,61.235,-92.577,168.928,41.696,157.815
C01376=1034.115,60.985,-92.559,168.926,41.697,157.815
C01377=1034.108,60.699,-92.539,168.923,41.697,157.815
C01378=1034.100,60.413,-92.520,168.920,41.698,157.815
C01379=1034.093,60.127,-92.500,168.918,41.699,157.815
C01380=1034.086,59.841,-92.480,168.915,41.700,157.815
C01381=1034.079,59.592,-92.462,168.913,41.700,157.815
C01382=1034.073,59.342,-92.445,168.911,41.701,157.815
C01383=1034.067,59.093,-92.428,168.909,41.702,157.815
C01384=1034.060,58.844,-92.410,168.907,41.703,157.815
C01385=1034.054,58.594,-92.392,168.905,41.704,157.815
C01386=1034.048,58.345,-92.375,168.902,41.705,157.815
C01387=1034.041,58.096,-92.358,168.900,41.705,157.815
C01388=1034.036,57.846,-92.341,168.898,41.706,157.815
C01389=1034.029,57.597,-92.324,168.895,41.707,157.815
C01390=1034.022,57.347,-92.306,168.893,41.707,157.815
C01391=1034.016,57.098,-92.289,168.891,41.708,157.815
C01392=1034.010,56.849,-92.272,168.889,41.709,157.815
C01393=1034.003,56.600,-92.255,168.886,41.709,157.815
C01394=1033.996,56.351,-92.237,168.884,41.710,157.815
C01395=1033.990,56.101,-92.219,168.883,41.711,157.815
C01396=1033.984,55.852,-92.202,168.880,41.712,157.815
C01397=1033.977,55.602,-92.186,168.878,41.713,157.815
C01398=1033.972,55.353,-92.168,168.876,41.713,157.815
C01399=1033.965,55.104,-92.151,168.873,41.714,157.815
C01400=1033.958,54.854,-92.133,168.871,41.715,157.815
C01401=1033.953,54.605,-92.116,168.869,41.715,157.815
C01402=1033.946,54.356,-92.099,168.867,41.716,157.815
C01403=1033.940,54.106,-92.082,168.864,41.717,157.815
C01404=1033.934,53.857,-92.064,168.862,41.717,157.815
C01405=1033.928,53.608,-92.047,168.860,41.718,157.815
C01406=1033.921,53.359,-92.030,168.857,41.719,157.815
C01407=1033.915,53.110,-92.013,168.855,41.720,157.815
C01408=1033.909,52.859,-91.996,168.854,41.721,157.815
C01409=1033.902,52.611,-91.979,168.852,41.721,157.815
C01410=1033.895,52.361,-91.962,168.849,41.722,157.815
C01411=1033.890,52.112,-91.944,168.847,41.722,157.815
C01412=1033.883,51.862,-91.927,168.845,41.723,157.815
C01413=1033.877,51.614,-91.910,168.842,41.724,157.815
C01414=1033.871,51.364,-91.892,168.840,41.724,157.815
C01415=1033.865,51.115,-91.876,168.838,41.725,157.815
C01416=1033.858,50.865,-91.859,168.836,41.726,157.815
C01417=1033.853,50.616,-91.841,168.833,41.727,157.815
C01418=1033.846,50.367,-91.824,168.831,41.727,157.815
C01419=1033.840,50.118,-91.807,168.829,41.728,157.815
C01420=1033.833,49.868,-91.790,168.826,41.729,157.815
C01421=1033.828,49.619,-91.773,168.824,41.729,157.815
C01422=1033.821,49.369,-91.755,168.823,41.730,157.815
C01423=1033.815,49.120,-91.739,168.820,41.730,157.815
C01424=1033.809,48.870,-91.721,168.818,41.731,157.815
C01425=1033.802,48.621,-91.704,168.816,41.732,157.815
C01426=1033.796,48.372,-91.688,168.814,41.733,157.815
C01427=1033.790,48.123,-91.671,168.812,41.734,157.815
C01428=1033.784,47.874,-91.653,168.809,41.734,157.815
C01429=1033.777,47.624,-91.637,168.807,41.735,157.815
C01430=1033.771,47.375,-91.620,168.805,41.735,157.815
C01431=1033.765,47.125,-91.603,168.802,41.736,157.815
C01432=1033.759,46.876,-91.585,168.800,41.737,157.815
C01433=1033.753,46.627,-91.568,168.798,41.737,157.815
C01434=1033.746,46.377,-91.552,168.796,41.738,157.815
C01435=1033.741,46.128,-91.534,168.793,41.739,157.815
C01436=1033.734,45.878,-91.518,168.791,41.739,157.815
C01437=1033.728,45.629,-91.501,168.789,41.740,157.815
C01438=1033.722,45.380,-91.484,168.787,41.740,157.815
C01439=1033.716,45.130,-91.466,168.785,41.741,157.815
C01440=1033.710,44.881,-91.449,168.783,41.742,157.815
C01441=1033.703,44.595,-91.430,168.780,41.743,157.815
C01442=1033.695,44.309,-91.411,168.778,41.744,157.815
C01443=1033.688,44.022,-91.391,168.775,41.744,157.815
C01444=1033.681,43.735,-91.372,168.773,41.745,157.815
C01445=1033.675,43.487,-91.355,168.770,41.745,157.815
C01446=1033.669,43.237,-91.339,168.768,41.746,157.815
C01447=1033.663,42.988,-91.321,168.766,41.746,157.815
C01448=1033.657,42.738,-91.305,168.763,41.748,157.815
C01449=1033.650,42.489,-91.287,168.761,41.748,157.815
C01450=1033.644,42.239,-91.271,168.759,41.749,157.815
C01451=1033.638,41.990,-91.255,168.756,41.750,157.815
C01452=1033.631,41.741,-91.237,168.755,41.751,157.815
C01453=1033.626,41.491,-91.221,168.752,41.751,157.815
C01454=1033.619,41.243,-91.204,168.750,41.752,157.815
C01455=1033.613,40.992,-91.188,168.748,41.753,157.815
C01456=1033.607,40.743,-91.171,168.746,41.753,157.815
C01457=1033.600,40.494,-91.154,168.744,41.754,157.815
C01458=1033.594,40.244,-91.138,168.741,41.755,157.815
C01459=1033.588,39.995,-91.121,168.739,41.756,157.815
C01460=1033.581,39.746,-91.104,168.737,41.756,157.815
C01461=1033.575,39.496,-91.088,168.734,41.757,157.815
C01462=1033.569,39.247,-91.072,168.732,41.758,157.815
C01463=1033.563,38.998,-91.055,168.730,41.759,157.815
C01464=1033.556,38.748,-91.038,168.727,41.759,157.815
C01465=1033.550,38.499,-91.022,168.725,41.760,157.815
C01466=1033.543,38.250,-91.005,168.723,41.760,157.815
C01467=1033.537,38.000,-90.989,168.721,41.761,157.815
C01468=1033.531,37.751,-90.972,168.719,41.762,157.815
C01469=1033.525,37.502,-90.956,168.717,41.763,157.815
C01470=1033.518,37.252,-90.939,168.714,41.764,157.815
C01471=1033.512,37.003,-90.923,168.712,41.765,157.815
C01472=1033.506,36.753,-90.906,168.710,41.765,157.815
C01473=1033.500,36.503,-90.890,168.707,41.766,157.815
C01474=1033.494,36.254,-90.874,168.705,41.767,157.815
C01475=1033.487,36.006,-90.857,168.703,41.768,157.815
C01476=1033.480,35.756,-90.841,168.700,41.768,157.815
C01477=1033.474,35.506,-90.824,168.698,41.769,157.815
C01478=1033.468,35.257,-90.808,168.697,41.770,157.815
C01479=1033.462,35.008,-90.792,168.694,41.770,157.815
C01480=1033.455,34.758,-90.776,168.692,41.771,157.815
C01481=1033.449,34.509,-90.759,168.690,41.772,157.815
C01482=1033.443,34.260,-90.742,168.687,41.773,157.815
C01483=1033.436,34.011,-90.727,168.685,41.774,157.815
C01484=1033.430,33.761,-90.710,168.682,41.775,157.815
C01485=1033.424,33.511,-90.694,168.680,41.776,157.815
C01486=1033.418,33.262,-90.678,168.678,41.776,157.815
C01487=1033.410,33.012,-90.662,168.675,41.777,157.815
C01488=1033.404,32.763,-90.645,168.674,41.778,157.815
C01489=1033.399,32.514,-90.629,168.672,41.779,157.815
C01490=1033.393,32.264,-90.613,168.669,41.779,157.815
C01491=1033.386,32.015,-90.597,168.667,41.780,157.815
C01492=1033.379,31.766,-90.580,168.665,41.781,157.815
C01493=1033.373,31.516,-90.564,168.662,41.782,157.815
C01494=1033.366,31.267,-90.548,168.660,41.782,157.815
C01495=1033.360,31.018,-90.532,168.658,41.783,157.815
C01496=1033.354,30.768,-90.515,168.655,41.784,157.815
C01497=1033.348,30.519,-90.499,168.653,41.785,157.815
C01498=1033.341,30.270,-90.483,168.651,41.786,157.815
C01499=1033.335,30.020,-90.467,168.648,41.786,157.815
C01500=1033.329,29.771,-90.451,168.647,41.787,157.815
C01501=1033.323,29.522,-90.434,168.644,41.788,157.815
C01502=1033.316,29.272,-90.418,168.642,41.788,157.815
C01503=1033.310,29.022,-90.402,168.640,41.789,157.815
C01504=1033.304,28.773,-90.386,168.637,41.790,157.815
C01505=1033.297,28.486,-90.368,168.635,41.791,157.815
C01506=1033.290,28.200,-90.349,168.632,41.792,157.815
C01507=1033.282,27.914,-90.331,168.629,41.793,157.815
C01508=1033.275,27.627,-90.313,168.627,41.794,157.815
C01509=1033.269,27.378,-90.297,168.624,41.795,157.815
C01510=1033.263,27.128,-90.281,168.622,41.795,157.815
C01511=1033.257,26.879,-90.265,168.620,41.796,157.815
C01512=1033.250,26.630,-90.249,168.618,41.797,157.815
C01513=1033.244,26.381,-90.233,168.616,41.798,157.815
C01514=1033.237,26.131,-90.217,168.613,41.798,157.815
C01515=1033.231,25.881,-90.201,168.611,41.799,157.815
C01516=1033.224,25.632,-90.185,168.608,41.800,157.815
C01517=1033.218,25.383,-90.169,168.606,41.801,157.815
C01518=1033.212,25.134,-90.153,168.604,41.802,157.815
C01519=1033.206,24.884,-90.137,168.601,41.803,157.815
C01520=1033.199,24.635,-90.122,168.599,41.804,157.815
C01521=1033.193,24.385,-90.106,168.598,41.804,157.815
C01522=1033.186,24.136,-90.090,168.595,41.806,157.815
C01523=1033.180,23.886,-90.074,168.593,41.806,157.815
C01524=1033.174,23.637,-90.058,168.590,41.807,157.815
C01525=1033.168,23.387,-90.043,168.588,41.808,157.815
C01526=1033.161,23.138,-90.027,168.586,41.809,157.815
C01527=1033.155,22.889,-90.011,168.583,41.809,157.815
C01528=1033.149,22.639,-89.996,168.581,41.810,157.815
C01529=1033.143,22.390,-89.979,168.578,41.811,157.815
C01530=1033.136,22.140,-89.963,168.576,41.811,157.815
C01531=1033.130,21.891,-89.947,168.574,41.812,157.815
C01532=1033.123,21.641,-89.932,168.572,41.813,157.815
C01533=1033.117,21.392,-89.916,168.570,41.814,157.815
C01534=1033.111,21.143,-89.900,168.567,41.815,157.815
C01535=1033.105,20.893,-89.885,168.565,41.816,157.815
C01536=1033.098,20.644,-89.869,168.563,41.817,157.815
C01537=1033.092,20.395,-89.853,168.560,41.818,157.815
C01538=1033.086,20.145,-89.838,168.558,41.818,157.815
C01539=1033.079,19.896,-89.822,168.555,41.819,157.815
C01540=1033.073,19.646,-89.806,168.553,41.820,157.815
C01541=1033.067,19.397,-89.791,168.551,41.820,157.815
C01542=1033.061,19.147,-89.775,168.548,41.821,157.815
C01543=1033.055,18.898,-89.760,168.547,41.822,157.815
C01544=1033.048,18.649,-89.744,168.544,41.823,157.815
C01545=1033.042,18.399,-89.728,168.542,41.824,157.816
C01546=1033.036,18.150,-89.713,168.539,41.825,157.815
C01547=1033.029,17.900,-89.697,168.537,41.826,157.815
C01548=1033.023,17.651,-89.682,168.535,41.827,157.816
C01549=1033.016,17.401,-89.666,168.532,41.828,157.816
C01550=1033.010,17.151,-89.651,168.530,41.829,157.816
C01551=1033.004,16.902,-89.634,168.527,41.829,157.816
C01552=1032.997,16.652,-89.620,168.526,41.830,157.816
C01553=1032.991,16.403,-89.604,168.524,41.831,157.816
C01554=1032.984,16.153,-89.589,168.521,41.832,157.816
C01555=1032.978,15.904,-89.573,168.519,41.832,157.816
C01556=1032.972,15.655,-89.558,168.516,41.833,157.816
C01557=1032.966,15.406,-89.542,168.514,41.834,157.816
C01558=1032.960,15.156,-89.527,168.511,41.835,157.816
C01559=1032.953,14.907,-89.511,168.509,41.836,157.816
C01560=1032.947,14.657,-89.496,168.507,41.836,157.816
C01561=1032.941,14.408,-89.480,168.504,41.838,157.816
C01562=1032.935,14.158,-89.465,168.503,41.838,157.816
C01563=1032.928,13.909,-89.450,168.500,41.839,157.816
C01564=1032.922,13.659,-89.434,168.498,41.840,157.816
C01565=1032.916,13.410,-89.419,168.495,41.841,157.816
C01566=1032.910,13.160,-89.404,168.493,41.842,157.816
C01567=1032.903,12.911,-89.388,168.490,41.843,157.816
C01568=1032.897,12.661,-89.373,168.488,41.844,157.816
C01569=1032.889,12.376,-89.356,168.485,41.845,157.816
C01570=1032.881,12.091,-89.338,168.483,41.846,157.816
C01571=1032.875,11.806,-89.321,168.480,41.847,157.816
C01572=1032.867,11.521,-89.304,168.478,41.848,157.816
C01573=1032.860,11.272,-89.289,168.475,41.849,157.816
C01574=1032.854,11.022,-89.273,168.473,41.850,157.816
C01575=1032.848,10.772,-89.258,168.470,41.851,157.816
C01576=1032.841,10.523,-89.243,168.468,41.852,157.816
C01577=1032.835,10.274,-89.228,168.465,41.852,157.816
C01578=1032.828,10.024,-89.213,168.463,41.853,157.816
C01579=1032.822,9.774,-89.198,168.461,41.854,157.816
C01580=1032.816,9.525,-89.183,168.459,41.855,157.816
C01581=1032.810,9.276,-89.167,168.456,41.856,157.816
C01582=1032.803,9.027,-89.153,168.454,41.857,157.816
C01583=1032.797,8.777,-89.138,168.451,41.858,157.816
C01584=1032.790,8.527,-89.123,168.449,41.859,157.816
C01585=1032.784,8.278,-89.108,168.446,41.860,157.816
C01586=1032.777,8.029,-89.092,168.444,41.861,157.816
C01587=1032.771,7.779,-89.077,168.442,41.862,157.816
C01588=1032.765,7.529,-89.062,168.440,41.863,157.816
C01589=1032.759,7.280,-89.048,168.437,41.864,157.816
C01590=1032.752,7.031,-89.033,168.435,41.865,157.816
C01591=1032.746,6.781,-89.018,168.432,41.866,157.816
C01592=1032.739,6.532,-89.002,168.430,41.866,157.816
C01593=1032.733,6.282,-88.987,168.427,41.867,157.816
C01594=1032.727,6.033,-88.972,168.425,41.868,157.816
C01595=1032.720,5.783,-88.957,168.422,41.869,157.816
C01596=1032.714,5.534,-88.943,168.421,41.870,157.817
C01597=1032.708,5.284,-88.928,168.418,41.871,157.817
C01598=1032.702,5.035,-88.913,168.416,41.871,157.816
C01599=1032.695,4.785,-88.898,168.413,41.873,157.816
C01600=1032.689,4.535,-88.883,168.411,41.873,157.817
C01601=1032.682,4.286,-88.867,168.408,41.875,157.817
C01602=1032.676,4.037,-88.853,168.406,41.876,157.817
C01603=1032.670,3.788,-88.838,168.403,41.877,157.817
C01604=1032.664,3.538,-88.823,168.401,41.877,157.817
C01605=1032.657,3.288,-88.808,168.399,41.878,157.817
C01606=1032.651,3.040,-88.793,168.397,41.879,157.817
C01607=1032.645,2.790,-88.778,168.395,41.880,157.817
C01608=1032.639,2.540,-88.763,168.392,41.881,157.817
C01609=1032.632,2.291,-88.748,168.390,41.881,157.817
C01610=1032.626,2.041,-88.733,168.387,41.882,157.817
C01611=1032.620,1.792,-88.719,168.385,41.883,157.817
C01612=1032.614,1.542,-88.704,168.382,41.884,157.817
C01613=1032.607,1.293,-88.689,168.380,41.885,157.817
C01614=1032.601,1.043,-88.674,168.377,41.886,157.817
C01615=1032.595,0.794,-88.659,168.376,41.887,157.817
C01616=1032.589,0.544,-88.644,168.373,41.888,157.817
C01617=1032.582,0.295,-88.629,168.371,41.889,157.817
C01618=1032.577,0.046,-88.615,168.368,41.890,157.817
C01619=1032.570,-0.204,-88.600,168.366,41.890,157.817
C01620=1032.564,-0.454,-88.585,168.363,41.891,157.817
C01621=1032.557,-0.703,-88.570,168.361,41.892,157.817
C01622=1032.552,-0.952,-88.555,168.358,41.893,157.817
C01623=1032.546,-1.202,-88.541,168.356,41.893,157.817
C01624=1032.539,-1.452,-88.526,168.353,41.894,157.817
C01625=1032.533,-1.701,-88.512,168.352,41.895,157.817
C01626=1032.527,-1.951,-88.497,168.349,41.896,157.817
C01627=1032.521,-2.200,-88.482,168.347,41.897,157.817
C01628=1032.515,-2.449,-88.467,168.344,41.898,157.817
C01629=1032.509,-2.699,-88.452,168.342,41.899,157.817
C01630=1032.502,-2.949,-88.437,168.339,41.900,157.817
C01631=1032.496,-3.198,-88.423,168.337,41.901,157.817
C01632=1032.490,-3.448,-88.409,168.334,41.901,157.817
C01633=1032.484,-3.720,-88.392,168.331,41.902,157.817
C01634=1032.477,-3.993,-88.377,168.329,41.903,157.817
C01635=1032.469,-4.266,-88.361,168.327,41.904,157.817
C01636=1032.463,-4.538,-88.345,168.324,41.905,157.817
C01637=1032.456,-4.788,-88.331,168.321,41.906,157.817
C01638=1032.450,-5.038,-88.316,168.319,41.907,157.817
C01639=1032.444,-5.287,-88.301,168.316,41.908,157.817
C01640=1032.437,-5.537,-88.288,168.314,41.909,157.817
C01641=1032.430,-5.797,-88.272,168.311,41.910,157.817
C01642=1032.423,-6.056,-88.257,168.309,41.911,157.817
C01643=1032.417,-6.317,-88.242,168.307,41.912,157.817
C01644=1032.411,-6.577,-88.227,168.304,41.913,157.817
C01645=1032.404,-6.826,-88.213,168.301,41.915,157.817
C01646=1032.398,-7.076,-88.199,168.299,41.915,157.817
C01647=1032.392,-7.325,-88.184,168.296,41.917,157.817
C01648=1032.385,-7.575,-88.170,168.294,41.918,157.817
C01649=1032.379,-7.824,-88.156,168.291,41.919,157.817
C01650=1032.372,-8.073,-88.141,168.289,41.920,157.817
C01651=1032.367,-8.323,-88.128,168.287,41.921,157.817
C01652=1032.360,-8.573,-88.113,168.284,41.922,157.817
C01653=1032.353,-8.822,-88.098,168.282,41.923,157.818
C01654=1032.348,-9.072,-88.084,168.279,41.924,157.818
C01655=1032.341,-9.321,-88.069,168.277,41.925,157.818
C01656=1032.335,-9.571,-88.056,168.274,41.926,157.818
C01657=1032.329,-9.820,-88.041,168.272,41.927,157.818
C01658=1032.322,-10.070,-88.027,168.270,41.927,157.818
C01659=1032.316,-10.319,-88.013,168.267,41.928,157.818
C01660=1032.310,-10.569,-87.998,168.265,41.929,157.818
C01661=1032.303,-10.818,-87.985,168.262,41.930,157.818
C01662=1032.297,-11.068,-87.970,168.260,41.931,157.818
C01663=1032.291,-11.317,-87.957,168.257,41.932,157.818
C01664=1032.284,-11.567,-87.942,168.254,41.933,157.818
C01665=1032.279,-11.816,-87.928,168.253,41.934,157.818
C01666=1032.272,-12.066,-87.913,168.250,41.935,157.818
C01667=1032.266,-12.316,-87.899,168.248,41.936,157.818
C01668=1032.259,-12.564,-87.885,168.245,41.937,157.818
C01669=1032.253,-12.815,-87.871,168.242,41.938,157.818
C01670=1032.247,-13.064,-87.856,168.240,41.939,157.818
C01671=1032.241,-13.314,-87.843,168.237,41.940,157.818
C01672=1032.235,-13.563,-87.828,168.235,41.941,157.818
C01673=1032.228,-13.813,-87.815,168.232,41.942,157.818
C01674=1032.223,-14.062,-87.801,168.230,41.943,157.818
C01675=1032.216,-14.312,-87.786,168.228,41.944,157.818
C01676=1032.210,-14.561,-87.772,168.225,41.945,157.818
C01677=1032.204,-14.811,-87.758,168.223,41.946,157.818
C01678=1032.197,-15.060,-87.744,168.220,41.947,157.818
C01679=1032.191,-15.310,-87.730,168.217,41.947,157.818
C01680=1032.185,-15.559,-87.715,168.215,41.948,157.818
C01681=1032.179,-15.809,-87.702,168.212,41.949,157.818
C01682=1032.172,-16.058,-87.689,168.211,41.951,157.818
C01683=1032.166,-16.308,-87.674,168.208,41.952,157.818
C01684=1032.160,-16.557,-87.660,168.205,41.953,157.818
C01685=1032.153,-16.807,-87.647,168.203,41.954,157.818
C01686=1032.148,-17.057,-87.633,168.200,41.955,157.818
C01687=1032.140,-17.306,-87.618,168.197,41.956,157.818
C01688=1032.134,-17.556,-87.605,168.195,41.957,157.818
C01689=1032.128,-17.806,-87.591,168.193,41.958,157.818
C01690=1032.122,-18.055,-87.578,168.190,41.959,157.818
C01691=1032.115,-18.304,-87.564,168.188,41.960,157.818
C01692=1032.109,-18.554,-87.549,168.185,41.961,157.818
C01693=1032.103,-18.803,-87.536,168.182,41.962,157.819
C01694=1032.096,-19.053,-87.523,168.180,41.963,157.819
C01695=1032.091,-19.302,-87.508,168.177,41.965,157.819
C01696=1032.084,-19.552,-87.494,168.175,41.966,157.819
C01697=1032.077,-19.834,-87.479,168.172,41.967,157.819
C01698=1032.070,-20.115,-87.464,168.169,41.968,157.819
C01699=1032.063,-20.397,-87.447,168.166,41.970,157.819
C01700=1032.055,-20.678,-87.433,168.163,41.971,157.819
C01701=1032.050,-20.928,-87.419,168.161,41.972,157.819
C01702=1032.043,-21.178,-87.406,168.159,41.973,157.819
C01703=1032.036,-21.426,-87.392,168.156,41.974,157.819
C01704=1032.030,-21.677,-87.377,168.154,41.975,157.819
C01705=1032.024,-21.926,-87.364,168.151,41.976,157.819
C01706=1032.018,-22.175,-87.351,168.149,41.977,157.819
C01707=1032.012,-22.425,-87.337,168.146,41.978,157.819
C01708=1032.006,-22.675,-87.323,168.143,41.979,157.819
C01709=1031.999,-22.924,-87.310,168.142,41.980,157.819
C01710=1031.993,-23.174,-87.296,168.139,41.981,157.819
C01711=1031.987,-23.424,-87.283,168.136,41.982,157.819
C01712=1031.981,-23.673,-87.269,168.134,41.983,157.819
C01713=1031.974,-23.922,-87.255,168.131,41.984,157.819
C01714=1031.968,-24.172,-87.241,168.128,41.985,157.819
C01715=1031.962,-24.421,-87.228,168.126,41.986,157.819
C01716=1031.955,-24.671,-87.214,168.123,41.987,157.819
C01717=1031.950,-24.921,-87.200,168.121,41.988,157.819
C01718=1031.944,-25.170,-87.187,168.119,41.989,157.819
C01719=1031.937,-25.420,-87.173,168.116,41.990,157.819
C01720=1031.931,-25.669,-87.160,168.113,41.991,157.819
C01721=1031.925,-25.919,-87.146,168.111,41.992,157.819
C01722=1031.918,-26.169,-87.133,168.108,41.993,157.819
C01723=1031.912,-26.418,-87.119,168.105,41.994,157.819
C01724=1031.907,-26.667,-87.105,168.104,41.995,157.819
C01725=1031.900,-26.917,-87.092,168.101,41.996,157.819
C01726=1031.894,-27.167,-87.079,168.098,41.998,157.820
C01727=1031.888,-27.417,-87.066,168.095,41.999,157.820
C01728=1031.881,-27.666,-87.053,168.093,42.000,157.820
C01729=1031.875,-27.916,-87.039,168.090,42.001,157.820
C01730=1031.868,-28.165,-87.026,168.087,42.002,157.820
C01731=1031.862,-28.414,-87.013,168.085,42.003,157.820
C01732=1031.856,-28.664,-86.999,168.083,42.004,157.820
C01733=1031.849,-28.914,-86.986,168.080,42.006,157.820
C01734=1031.843,-29.163,-86.973,168.077,42.007,157.820
C01735=1031.837,-29.413,-86.960,168.075,42.008,157.820
C01736=1031.831,-29.662,-86.947,168.072,42.009,157.820
C01737=1031.825,-29.912,-86.932,168.069,42.010,157.820
C01738=1031.819,-30.161,-86.919,168.067,42.011,157.820
C01739=1031.813,-30.411,-86.907,168.065,42.012,157.820
C01740=1031.806,-30.661,-86.893,168.062,42.014,157.820
C01741=1031.800,-30.911,-86.880,168.059,42.015,157.820
C01742=1031.793,-31.160,-86.866,168.056,42.016,157.820
C01743=1031.788,-31.410,-86.854,168.054,42.017,157.820
C01744=1031.781,-31.659,-86.841,168.052,42.018,157.820
C01745=1031.775,-31.909,-86.827,168.049,42.019,157.820
C01746=1031.768,-32.158,-86.814,168.047,42.020,157.820
C01747=1031.762,-32.408,-86.801,168.044,42.021,157.820
C01748=1031.756,-32.657,-86.788,168.041,42.022,157.820
C01749=1031.750,-32.907,-86.775,168.038,42.024,157.820
C01750=1031.743,-33.157,-86.762,168.037,42.025,157.821
C01751=1031.737,-33.406,-86.748,168.034,42.026,157.821
C01752=1031.731,-33.656,-86.735,168.031,42.027,157.821
C01753=1031.725,-33.905,-86.722,168.028,42.028,157.821
C01754=1031.719,-34.155,-86.709,168.026,42.029,157.821
C01755=1031.713,-34.404,-86.696,168.023,42.030,157.821
C01756=1031.707,-34.654,-86.683,168.020,42.031,157.821
C01757=1031.700,-34.904,-86.670,168.018,42.032,157.821
C01758=1031.694,-35.153,-86.657,168.016,42.034,157.821
C01759=1031.688,-35.403,-86.644,168.013,42.035,157.821
C01760=1031.682,-35.652,-86.631,168.010,42.036,157.821
C01761=1031.675,-35.933,-86.617,168.007,42.037,157.821
C01762=1031.667,-36.214,-86.601,168.004,42.038,157.821
C01763=1031.660,-36.495,-86.587,168.001,42.039,157.821
C01764=1031.653,-36.775,-86.573,167.999,42.041,157.821
C01765=1031.647,-37.025,-86.560,167.996,42.042,157.821
C01766=1031.641,-37.275,-86.546,167.993,42.043,157.821
C01767=1031.635,-37.524,-86.534,167.990,42.044,157.821
C01768=1031.629,-37.774,-86.521,167.988,42.045,157.821
C01769=1031.622,-38.023,-86.507,167.985,42.046,157.821
C01770=1031.616,-38.273,-86.495,167.983,42.047,157.821
C01771=1031.610,-38.522,-86.482,167.980,42.048,157.821
C01772=1031.604,-38.772,-86.469,167.978,42.049,157.821
C01773=1031.598,-39.021,-86.456,167.975,42.051,157.821
C01774=1031.592,-39.271,-86.443,167.972,42.052,157.821
C01775=1031.586,-39.521,-86.431,167.969,42.053,157.821
C01776=1031.579,-39.770,-86.418,167.968,42.054,157.821
C01777=1031.573,-40.020,-86.405,167.965,42.056,157.822
C01778=1031.567,-40.270,-86.392,167.962,42.057,157.822
C01779=1031.560,-40.519,-86.380,167.959,42.058,157.822
C01780=1031.554,-40.769,-86.367,167.956,42.059,157.822
C01781=1031.548,-41.019,-86.354,167.954,42.061,157.822
C01782=1031.542,-41.268,-86.341,167.952,42.062,157.822
C01783=1031.535,-41.517,-86.329,167.949,42.063,157.822
C01784=1031.529,-41.767,-86.316,167.946,42.064,157.822
C01785=1031.523,-42.017,-86.304,167.943,42.066,157.822
C01786=1031.516,-42.266,-86.291,167.940,42.067,157.822
C01787=1031.510,-42.516,-86.278,167.939,42.068,157.822
C01788=1031.504,-42.766,-86.266,167.936,42.069,157.822
C01789=1031.498,-43.015,-86.253,167.933,42.070,157.822
C01790=1031.491,-43.265,-86.241,167.930,42.072,157.822
C01791=1031.486,-43.515,-86.228,167.927,42.073,157.822
C01792=1031.480,-43.764,-86.215,167.924,42.074,157.822
C01793=1031.473,-44.013,-86.203,167.923,42.075,157.822
C01794=1031.467,-44.263,-86.190,167.920,42.077,157.822
C01795=1031.461,-44.513,-86.178,167.917,42.078,157.822
C01796=1031.454,-44.762,-86.165,167.914,42.079,157.822
C01797=1031.448,-45.012,-86.152,167.911,42.080,157.822
C01798=1031.442,-45.262,-86.140,167.910,42.082,157.823
C01799=1031.436,-45.512,-86.127,167.907,42.083,157.823
